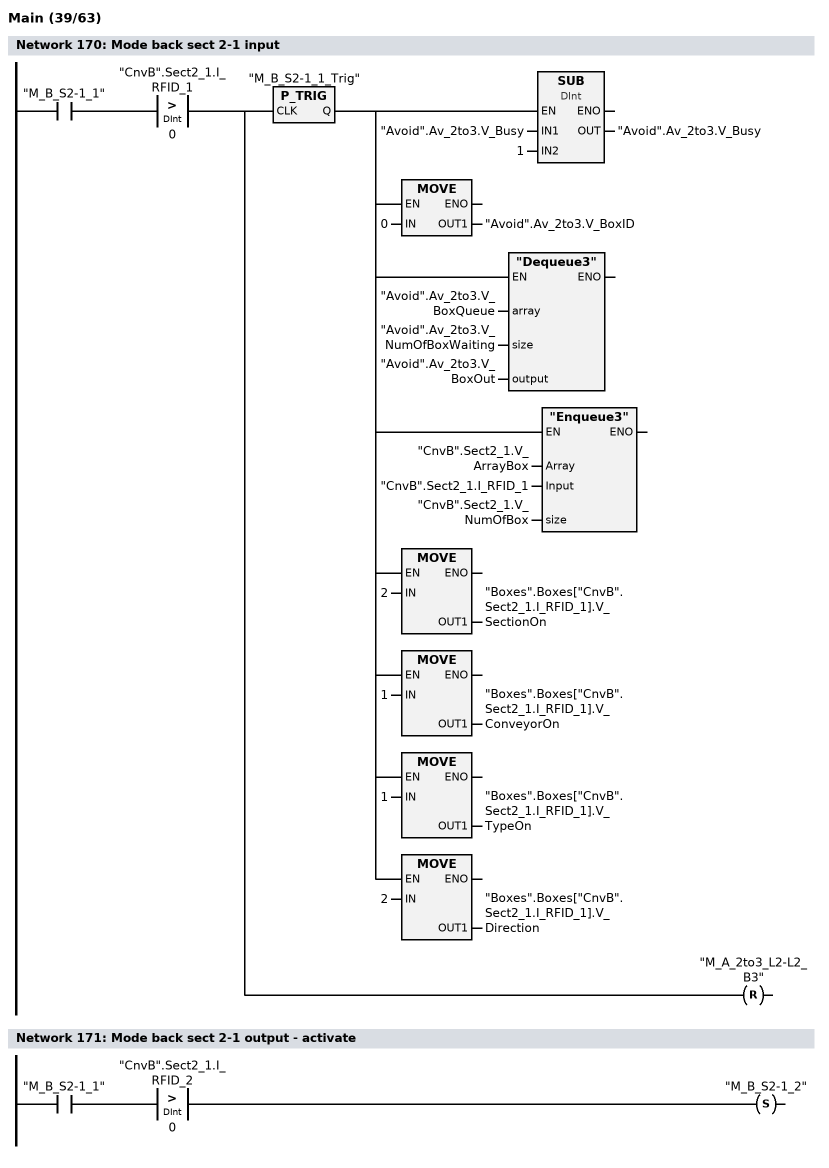
   RUNG wire#powerrail
      Contact( "M_B_S2-1_1" )
      { S7_Templates := "SrcType := DInt" } GT_Contact(in1 := "CnvB".Sect2_1.I_RFID_1, in2 := 0)
      wire#w1
      P_Trig( "M_B_S2-1_1_Trig" )
      wire#w2
      { S7_Templates := "SrcType := DInt" } Sub(in1 := "Avoid".Av_2to3.V_Busy, in2 := 1, out => "Avoid".Av_2to3.V_Busy)
   END_RUNG
   RUNG wire#w2
      Move(in := 0, out1 => "Avoid".Av_2to3.V_BoxID)
   END_RUNG
   RUNG wire#w2
      "Dequeue3"("array" := "Avoid".Av_2to3.V_BoxQueue, size := "Avoid".Av_2to3.V_NumOfBoxWaiting, output := "Avoid".Av_2to3.V_BoxOut)
   END_RUNG
   RUNG wire#w2
      "Enqueue3"("Array" := "CnvB".Sect2_1.V_ArrayBox, Input := "CnvB".Sect2_1.I_RFID_1, size := "CnvB".Sect2_1.V_NumOfBox)
   END_RUNG
   RUNG wire#w2
      Move(in := 2, out1 => "Boxes".Boxes["CnvB".Sect2_1.I_RFID_1].V_SectionOn)
   END_RUNG
   RUNG wire#w2
      Move(in := 1, out1 => "Boxes".Boxes["CnvB".Sect2_1.I_RFID_1].V_ConveyorOn)
   END_RUNG
   RUNG wire#w2
      Move(in := 1, out1 => "Boxes".Boxes["CnvB".Sect2_1.I_RFID_1].V_TypeOn)
   END_RUNG
   RUNG wire#w2
      Move(in := 2, out1 => "Boxes".Boxes["CnvB".Sect2_1.I_RFID_1].V_Direction)
   END_RUNG
   RUNG wire#w1
      R_Coil( "M_A_2to3_L2-L2_B3" )
   END_RUNG
   // the same network as SCL:
   #_w1 := "M_B_S2-1_1" AND ("CnvB".Sect2_1.I_RFID_1 > 0);
   #_w2 := #_w1 AND NOT "M_B_S2-1_1_Trig";   // rising edge
   "M_B_S2-1_1_Trig" := #_w1;
   IF #_w2 THEN
       "Avoid".Av_2to3.V_Busy := "Avoid".Av_2to3.V_Busy - 1;
       "Avoid".Av_2to3.V_BoxID := 0;
       "Dequeue3"("array" := "Avoid".Av_2to3.V_BoxQueue,
                  size := "Avoid".Av_2to3.V_NumOfBoxWaiting,
                  output := "Avoid".Av_2to3.V_BoxOut);
       "Enqueue3"("Array" := "CnvB".Sect2_1.V_ArrayBox,
                  Input := "CnvB".Sect2_1.I_RFID_1,
                  size := "CnvB".Sect2_1.V_NumOfBox);
       "Boxes".Boxes["CnvB".Sect2_1.I_RFID_1].V_SectionOn := 2;
       "Boxes".Boxes["CnvB".Sect2_1.I_RFID_1].V_ConveyorOn := 1;
       "Boxes".Boxes["CnvB".Sect2_1.I_RFID_1].V_TypeOn := 1;
       "Boxes".Boxes["CnvB".Sect2_1.I_RFID_1].V_Direction := 2;
   END_IF;
   IF #_w1 THEN "M_A_2to3_L2-L2_B3" := FALSE; END_IF;
END_REGION

REGION Network 171: Mode back sect 2-1 output - activate
   RUNG wire#powerrail
      Contact( "M_B_S2-1_1" )
      { S7_Templates := "SrcType := DInt" } GT_Contact(in1 := "CnvB".Sect2_1.I_RFID_2, in2 := 0)
      S_Coil( "M_B_S2-1_2" )
   END_RUNG
   // the same network as SCL:
   IF "M_B_S2-1_1" AND ("CnvB".Sect2_1.I_RFID_2 > 0) THEN "M_B_S2-1_2" := TRUE; END_IF;
END_REGION

REGION Network 172: Mode back sect 2-1 output
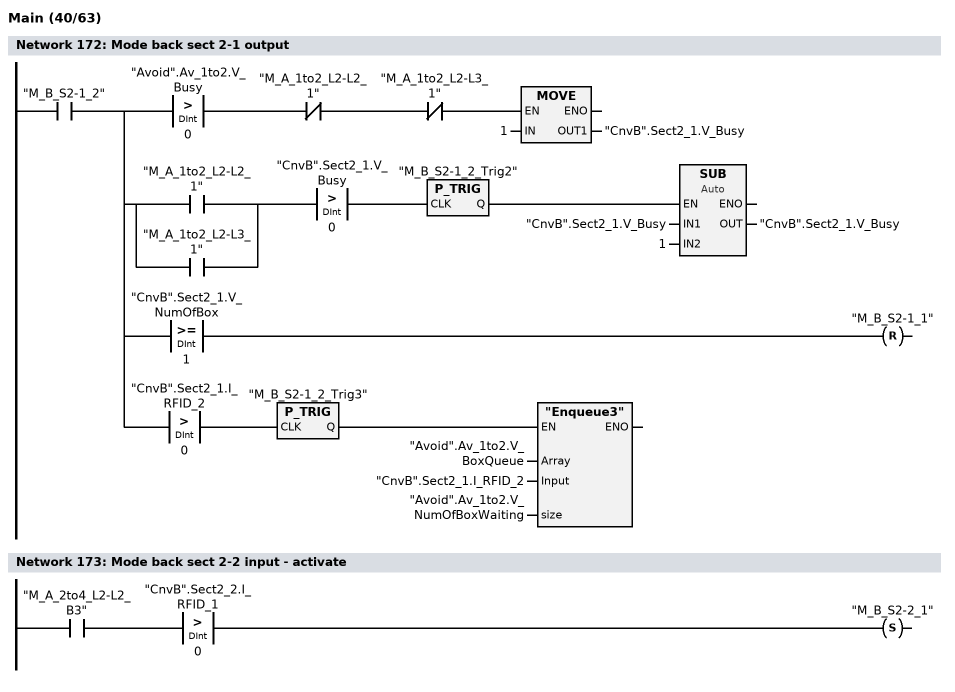
   RUNG wire#powerrail
      Contact( "M_B_S2-1_2" )
      wire#w1
      { S7_Templates := "SrcType := DInt" } GT_Contact(in1 := "Avoid".Av_1to2.V_Busy, in2 := 0)
      I_Contact( "M_A_1to2_L2-L2_1" )
      I_Contact( "M_A_1to2_L2-L3_1" )
      Move(in := 1, out1 => "CnvB".Sect2_1.V_Busy)
   END_RUNG
   RUNG wire#w1
      Contact( "M_A_1to2_L2-L2_1" )
      wire#w2
      { S7_Templates := "SrcType := DInt" } GT_Contact(in1 := "CnvB".Sect2_1.V_Busy, in2 := 0)
      P_Trig( "M_B_S2-1_2_Trig2" )
      Sub(in1 := "CnvB".Sect2_1.V_Busy, in2 := 1, out => "CnvB".Sect2_1.V_Busy)
   END_RUNG
   RUNG wire#w1
      Contact( "M_A_1to2_L2-L3_1" )
   END_RUNG wire#w2
   RUNG wire#w1
      { S7_Templates := "SrcType := DInt" } GE_Contact(in1 := "CnvB".Sect2_1.V_NumOfBox, in2 := 1)
      R_Coil( "M_B_S2-1_1" )
   END_RUNG
   RUNG wire#w1
      { S7_Templates := "SrcType := DInt" } GT_Contact(in1 := "CnvB".Sect2_1.I_RFID_2, in2 := 0)
      P_Trig( "M_B_S2-1_2_Trig3" )
      "Enqueue3"("Array" := "Avoid".Av_1to2.V_BoxQueue, Input := "CnvB".Sect2_1.I_RFID_2, size := "Avoid".Av_1to2.V_NumOfBoxWaiting)
   END_RUNG
   // the same network as SCL:
   IF "M_B_S2-1_2" AND ("Avoid".Av_1to2.V_Busy > 0) AND NOT "M_A_1to2_L2-L2_1" AND NOT "M_A_1to2_L2-L3_1" THEN
       "CnvB".Sect2_1.V_Busy := 1;
   END_IF;
   #_w1 := "M_B_S2-1_2" AND ("M_A_1to2_L2-L2_1" OR "M_A_1to2_L2-L3_1") AND ("CnvB".Sect2_1.V_Busy > 0);
   #_w2 := #_w1 AND NOT "M_B_S2-1_2_Trig2";   // rising edge
   "M_B_S2-1_2_Trig2" := #_w1;
   IF #_w2 THEN "CnvB".Sect2_1.V_Busy := "CnvB".Sect2_1.V_Busy - 1; END_IF;
   IF "M_B_S2-1_2" AND ("CnvB".Sect2_1.V_NumOfBox >= 1) THEN "M_B_S2-1_1" := FALSE; END_IF;
   #_w3 := "M_B_S2-1_2" AND ("CnvB".Sect2_1.I_RFID_2 > 0);
   #_w4 := #_w3 AND NOT "M_B_S2-1_2_Trig3";   // rising edge
   "M_B_S2-1_2_Trig3" := #_w3;
   IF #_w4 THEN
       "Enqueue3"("Array" := "Avoid".Av_1to2.V_BoxQueue,
                  Input := "CnvB".Sect2_1.I_RFID_2,
                  size := "Avoid".Av_1to2.V_NumOfBoxWaiting);
   END_IF;
END_REGION

REGION Network 173: Mode back sect 2-2 input - activate
   RUNG wire#powerrail
      Contact( "M_A_2to4_L2-L2_B3" )
      { S7_Templates := "SrcType := DInt" } GT_Contact(in1 := "CnvB".Sect2_2.I_RFID_1, in2 := 0)
      S_Coil( "M_B_S2-2_1" )
   END_RUNG
   // the same network as SCL:
   IF "M_A_2to4_L2-L2_B3" AND ("CnvB".Sect2_2.I_RFID_1 > 0) THEN "M_B_S2-2_1" := TRUE; END_IF;
END_REGION

REGION Network 174: Mode back sect 2-2 input
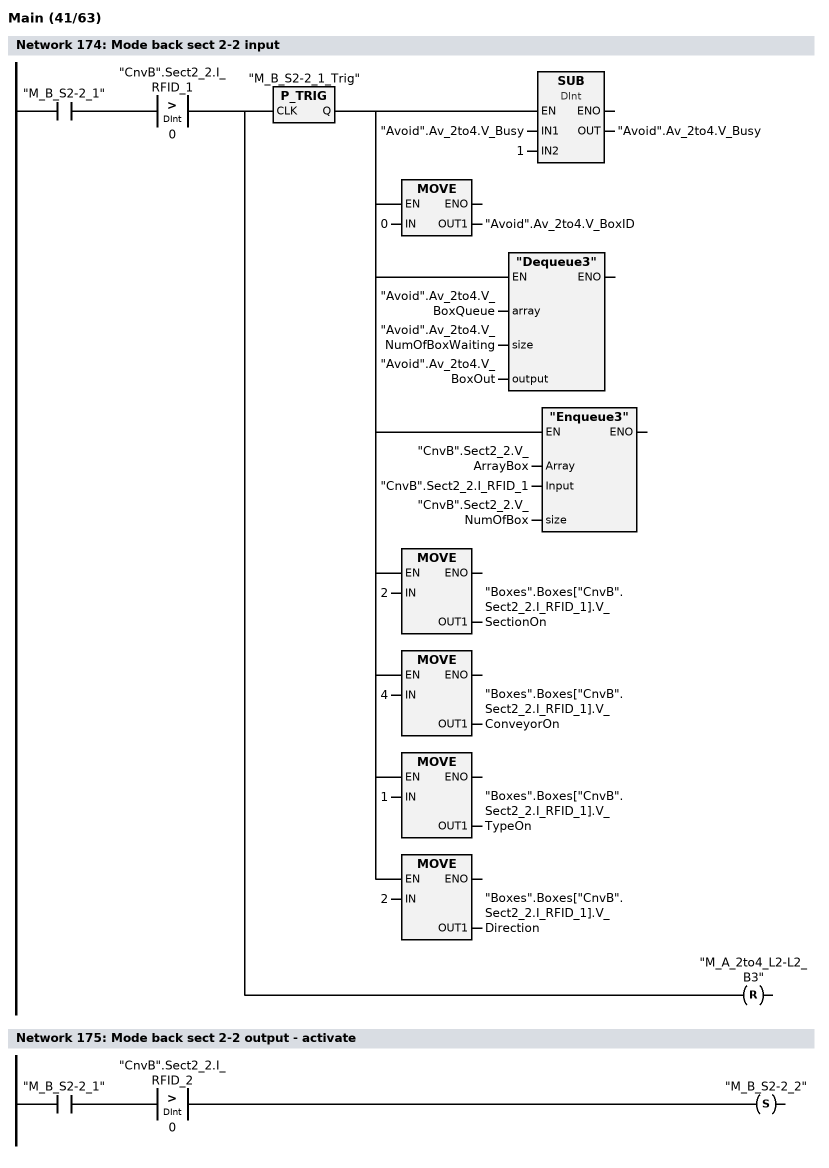
   RUNG wire#powerrail
      Contact( "M_B_S2-2_1" )
      { S7_Templates := "SrcType := DInt" } GT_Contact(in1 := "CnvB".Sect2_2.I_RFID_1, in2 := 0)
      wire#w1
      P_Trig( "M_B_S2-2_1_Trig" )
      wire#w2
      { S7_Templates := "SrcType := DInt" } Sub(in1 := "Avoid".Av_2to4.V_Busy, in2 := 1, out => "Avoid".Av_2to4.V_Busy)
   END_RUNG
   RUNG wire#w2
      Move(in := 0, out1 => "Avoid".Av_2to4.V_BoxID)
   END_RUNG
   RUNG wire#w2
      "Dequeue3"("array" := "Avoid".Av_2to4.V_BoxQueue, size := "Avoid".Av_2to4.V_NumOfBoxWaiting, output := "Avoid".Av_2to4.V_BoxOut)
   END_RUNG
   RUNG wire#w2
      "Enqueue3"("Array" := "CnvB".Sect2_2.V_ArrayBox, Input := "CnvB".Sect2_2.I_RFID_1, size := "CnvB".Sect2_2.V_NumOfBox)
   END_RUNG
   RUNG wire#w2
      Move(in := 2, out1 => "Boxes".Boxes["CnvB".Sect2_2.I_RFID_1].V_SectionOn)
   END_RUNG
   RUNG wire#w2
      Move(in := 4, out1 => "Boxes".Boxes["CnvB".Sect2_2.I_RFID_1].V_ConveyorOn)
   END_RUNG
   RUNG wire#w2
      Move(in := 1, out1 => "Boxes".Boxes["CnvB".Sect2_2.I_RFID_1].V_TypeOn)
   END_RUNG
   RUNG wire#w2
      Move(in := 2, out1 => "Boxes".Boxes["CnvB".Sect2_2.I_RFID_1].V_Direction)
   END_RUNG
   RUNG wire#w1
      R_Coil( "M_A_2to4_L2-L2_B3" )
   END_RUNG
   // the same network as SCL:
   #_w1 := "M_B_S2-2_1" AND ("CnvB".Sect2_2.I_RFID_1 > 0);
   #_w2 := #_w1 AND NOT "M_B_S2-2_1_Trig";   // rising edge
   "M_B_S2-2_1_Trig" := #_w1;
   IF #_w2 THEN
       "Avoid".Av_2to4.V_Busy := "Avoid".Av_2to4.V_Busy - 1;
       "Avoid".Av_2to4.V_BoxID := 0;
       "Dequeue3"("array" := "Avoid".Av_2to4.V_BoxQueue,
                  size := "Avoid".Av_2to4.V_NumOfBoxWaiting,
                  output := "Avoid".Av_2to4.V_BoxOut);
       "Enqueue3"("Array" := "CnvB".Sect2_2.V_ArrayBox,
                  Input := "CnvB".Sect2_2.I_RFID_1,
                  size := "CnvB".Sect2_2.V_NumOfBox);
       "Boxes".Boxes["CnvB".Sect2_2.I_RFID_1].V_SectionOn := 2;
       "Boxes".Boxes["CnvB".Sect2_2.I_RFID_1].V_ConveyorOn := 4;
       "Boxes".Boxes["CnvB".Sect2_2.I_RFID_1].V_TypeOn := 1;
       "Boxes".Boxes["CnvB".Sect2_2.I_RFID_1].V_Direction := 2;
   END_IF;
   IF #_w1 THEN "M_A_2to4_L2-L2_B3" := FALSE; END_IF;
END_REGION

REGION Network 175: Mode back sect 2-2 output - activate
   RUNG wire#powerrail
      Contact( "M_B_S2-2_1" )
      { S7_Templates := "SrcType := DInt" } GT_Contact(in1 := "CnvB".Sect2_2.I_RFID_2, in2 := 0)
      S_Coil( "M_B_S2-2_2" )
   END_RUNG
   // the same network as SCL:
   IF "M_B_S2-2_1" AND ("CnvB".Sect2_2.I_RFID_2 > 0) THEN "M_B_S2-2_2" := TRUE; END_IF;
END_REGION

REGION Network 176: Mode back sect 2-2 output
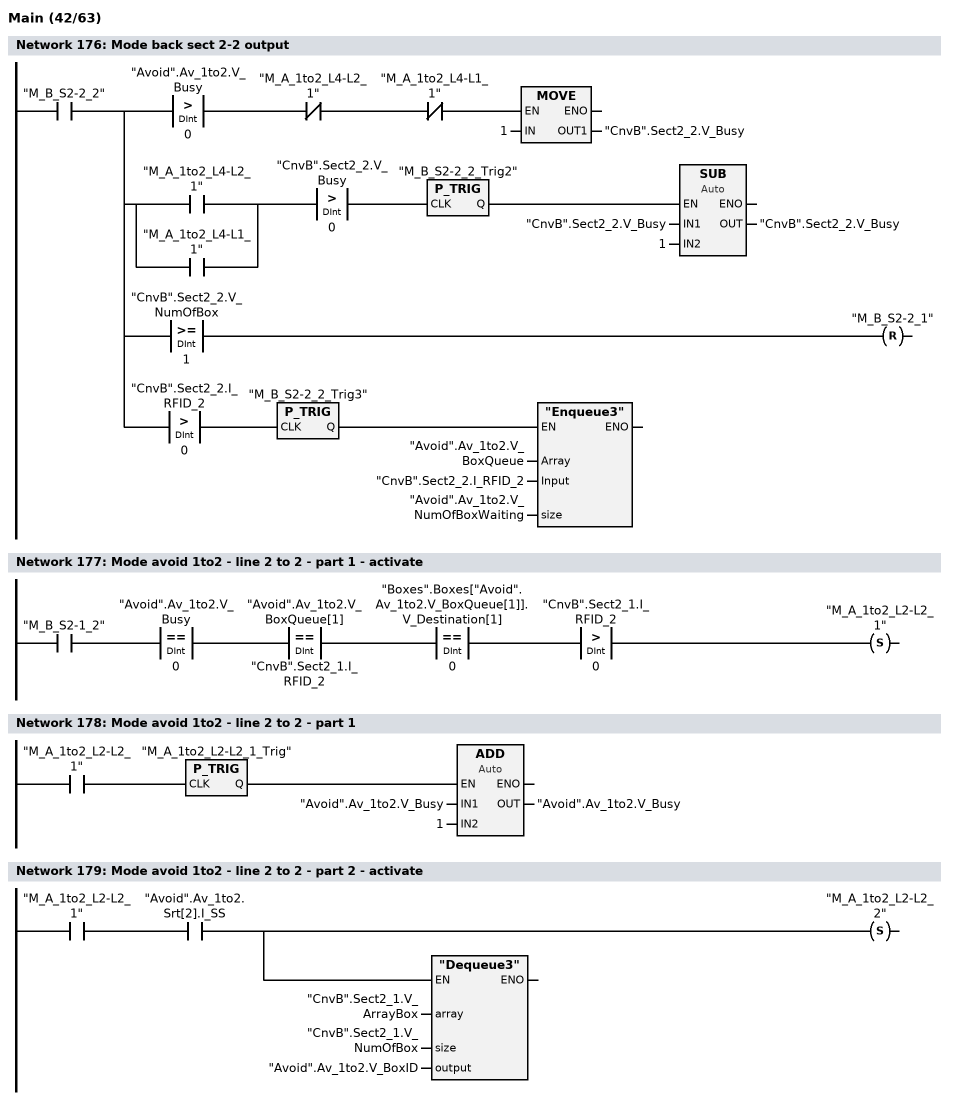
   RUNG wire#powerrail
      Contact( "M_B_S2-2_2" )
      wire#w1
      { S7_Templates := "SrcType := DInt" } GT_Contact(in1 := "Avoid".Av_1to2.V_Busy, in2 := 0)
      I_Contact( "M_A_1to2_L4-L2_1" )
      I_Contact( "M_A_1to2_L4-L1_1" )
      Move(in := 1, out1 => "CnvB".Sect2_2.V_Busy)
   END_RUNG
   RUNG wire#w1
      Contact( "M_A_1to2_L4-L2_1" )
      wire#w2
      { S7_Templates := "SrcType := DInt" } GT_Contact(in1 := "CnvB".Sect2_2.V_Busy, in2 := 0)
      P_Trig( "M_B_S2-2_2_Trig2" )
      Sub(in1 := "CnvB".Sect2_2.V_Busy, in2 := 1, out => "CnvB".Sect2_2.V_Busy)
   END_RUNG
   RUNG wire#w1
      Contact( "M_A_1to2_L4-L1_1" )
   END_RUNG wire#w2
   RUNG wire#w1
      { S7_Templates := "SrcType := DInt" } GE_Contact(in1 := "CnvB".Sect2_2.V_NumOfBox, in2 := 1)
      R_Coil( "M_B_S2-2_1" )
   END_RUNG
   RUNG wire#w1
      { S7_Templates := "SrcType := DInt" } GT_Contact(in1 := "CnvB".Sect2_2.I_RFID_2, in2 := 0)
      P_Trig( "M_B_S2-2_2_Trig3" )
      "Enqueue3"("Array" := "Avoid".Av_1to2.V_BoxQueue, Input := "CnvB".Sect2_2.I_RFID_2, size := "Avoid".Av_1to2.V_NumOfBoxWaiting)
   END_RUNG
   // the same network as SCL:
   IF "M_B_S2-2_2" AND ("Avoid".Av_1to2.V_Busy > 0) AND NOT "M_A_1to2_L4-L2_1" AND NOT "M_A_1to2_L4-L1_1" THEN
       "CnvB".Sect2_2.V_Busy := 1;
   END_IF;
   #_w1 := "M_B_S2-2_2" AND ("M_A_1to2_L4-L2_1" OR "M_A_1to2_L4-L1_1") AND ("CnvB".Sect2_2.V_Busy > 0);
   #_w2 := #_w1 AND NOT "M_B_S2-2_2_Trig2";   // rising edge
   "M_B_S2-2_2_Trig2" := #_w1;
   IF #_w2 THEN "CnvB".Sect2_2.V_Busy := "CnvB".Sect2_2.V_Busy - 1; END_IF;
   IF "M_B_S2-2_2" AND ("CnvB".Sect2_2.V_NumOfBox >= 1) THEN "M_B_S2-2_1" := FALSE; END_IF;
   #_w3 := "M_B_S2-2_2" AND ("CnvB".Sect2_2.I_RFID_2 > 0);
   #_w4 := #_w3 AND NOT "M_B_S2-2_2_Trig3";   // rising edge
   "M_B_S2-2_2_Trig3" := #_w3;
   IF #_w4 THEN
       "Enqueue3"("Array" := "Avoid".Av_1to2.V_BoxQueue,
                  Input := "CnvB".Sect2_2.I_RFID_2,
                  size := "Avoid".Av_1to2.V_NumOfBoxWaiting);
   END_IF;
END_REGION

REGION Network 177: Mode avoid 1to2 - line 2 to 2 - part 1 - activate
   RUNG wire#powerrail
      Contact( "M_B_S2-1_2" )
      { S7_Templates := "SrcType := DInt" } EQ_Contact(in1 := "Avoid".Av_1to2.V_Busy, in2 := 0)
      { S7_Templates := "SrcType := DInt" } EQ_Contact(in1 := "Avoid".Av_1to2.V_BoxQueue[1], in2 := "CnvB".Sect2_1.I_RFID_2)
      { S7_Templates := "SrcType := DInt" } EQ_Contact(in1 := "Boxes".Boxes["Avoid".Av_1to2.V_BoxQueue[1]].V_Destination[1], in2 := 0)
      { S7_Templates := "SrcType := DInt" } GT_Contact(in1 := "CnvB".Sect2_1.I_RFID_2, in2 := 0)
      S_Coil( "M_A_1to2_L2-L2_1" )
   END_RUNG
   // the same network as SCL:
   IF "M_B_S2-1_2" AND ("Avoid".Av_1to2.V_Busy = 0) AND ("Avoid".Av_1to2.V_BoxQueue[1] = "CnvB".Sect2_1.I_RFID_2) AND ("Boxes".Boxes["Avoid".Av_1to2.V_BoxQueue[1]].V_Destination[1] = 0) AND ("CnvB".Sect2_1.I_RFID_2 > 0) THEN
       "M_A_1to2_L2-L2_1" := TRUE;
   END_IF;
END_REGION

REGION Network 178: Mode avoid 1to2 - line 2 to 2 - part 1
   RUNG wire#powerrail
      Contact( "M_A_1to2_L2-L2_1" )
      P_Trig( "M_A_1to2_L2-L2_1_Trig" )
      Add(in1 := "Avoid".Av_1to2.V_Busy, in2 := 1, out => "Avoid".Av_1to2.V_Busy)
   END_RUNG
   // the same network as SCL:
   #_w1 := "M_A_1to2_L2-L2_1" AND NOT "M_A_1to2_L2-L2_1_Trig";   // rising edge
   "M_A_1to2_L2-L2_1_Trig" := "M_A_1to2_L2-L2_1";
   IF #_w1 THEN "Avoid".Av_1to2.V_Busy := "Avoid".Av_1to2.V_Busy + 1; END_IF;
END_REGION

REGION Network 179: Mode avoid 1to2 - line 2 to 2 - part 2 - activate
   RUNG wire#powerrail
      Contact( "M_A_1to2_L2-L2_1" )
      Contact( "Avoid".Av_1to2.Srt[2].I_SS )
      wire#w1
      S_Coil( "M_A_1to2_L2-L2_2" )
   END_RUNG
   RUNG wire#w1
      "Dequeue3"("array" := "CnvB".Sect2_1.V_ArrayBox, size := "CnvB".Sect2_1.V_NumOfBox, output := "Avoid".Av_1to2.V_BoxID)
   END_RUNG
   // the same network as SCL:
   IF "M_A_1to2_L2-L2_1" AND "Avoid".Av_1to2.Srt[2].I_SS THEN
       "M_A_1to2_L2-L2_2" := TRUE;
       "Dequeue3"("array" := "CnvB".Sect2_1.V_ArrayBox,
                  size := "CnvB".Sect2_1.V_NumOfBox,
                  output := "Avoid".Av_1to2.V_BoxID);
   END_IF;
END_REGION

REGION Network 180: Mode avoid 1to2 - line 2 to 2 - part 2
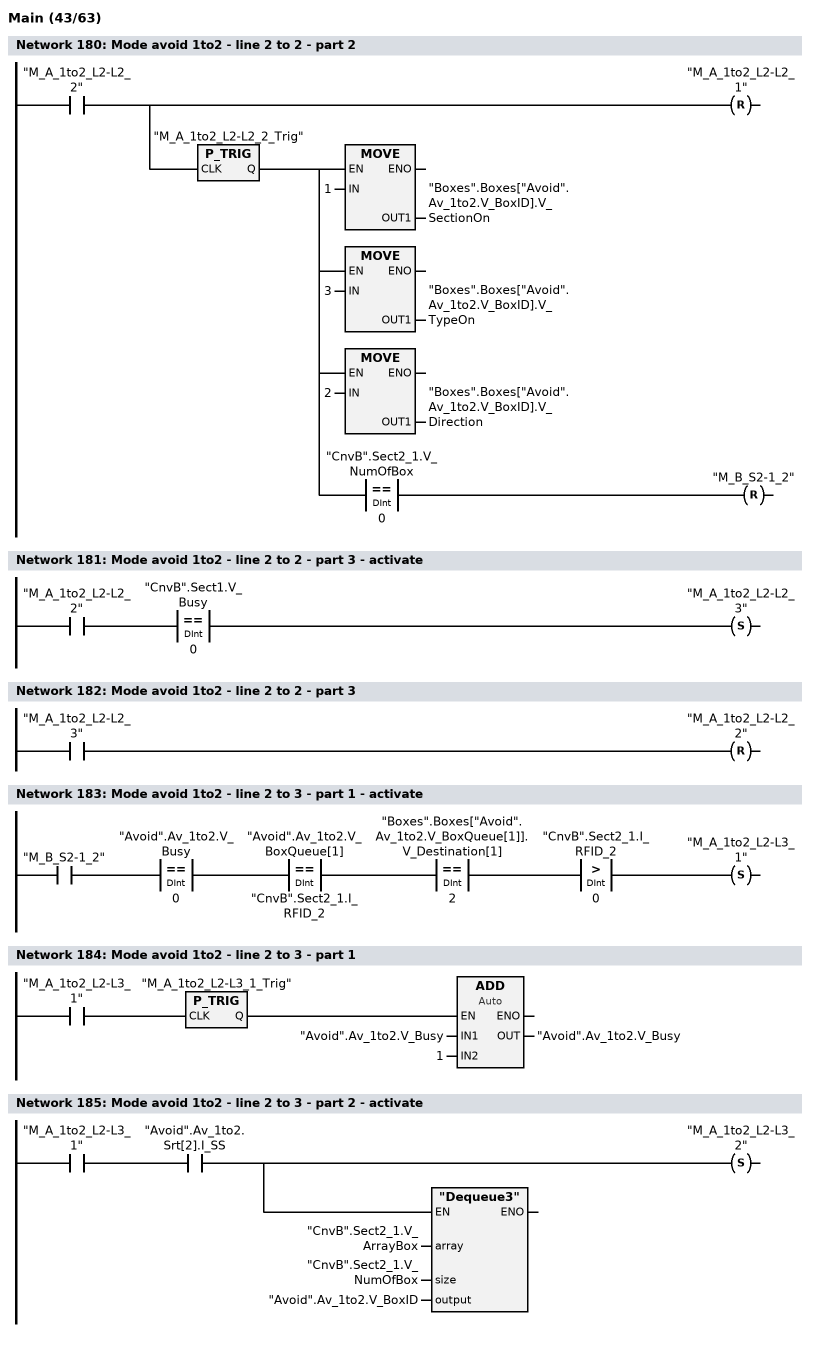
   RUNG wire#powerrail
      Contact( "M_A_1to2_L2-L2_2" )
      wire#w1
      R_Coil( "M_A_1to2_L2-L2_1" )
   END_RUNG
   RUNG wire#w1
      P_Trig( "M_A_1to2_L2-L2_2_Trig" )
      wire#w2
      Move(in := 1, out1 => "Boxes".Boxes["Avoid".Av_1to2.V_BoxID].V_SectionOn)
   END_RUNG
   RUNG wire#w2
      Move(in := 3, out1 => "Boxes".Boxes["Avoid".Av_1to2.V_BoxID].V_TypeOn)
   END_RUNG
   RUNG wire#w2
      Move(in := 2, out1 => "Boxes".Boxes["Avoid".Av_1to2.V_BoxID].V_Direction)
   END_RUNG
   RUNG wire#w2
      { S7_Templates := "SrcType := DInt" } EQ_Contact(in1 := "CnvB".Sect2_1.V_NumOfBox, in2 := 0)
      R_Coil( "M_B_S2-1_2" )
   END_RUNG
   // the same network as SCL:
   IF "M_A_1to2_L2-L2_2" THEN "M_A_1to2_L2-L2_1" := FALSE; END_IF;
   #_w1 := "M_A_1to2_L2-L2_2" AND NOT "M_A_1to2_L2-L2_2_Trig";   // rising edge
   "M_A_1to2_L2-L2_2_Trig" := "M_A_1to2_L2-L2_2";
   IF #_w1 THEN
       "Boxes".Boxes["Avoid".Av_1to2.V_BoxID].V_SectionOn := 1;
       "Boxes".Boxes["Avoid".Av_1to2.V_BoxID].V_TypeOn := 3;
       "Boxes".Boxes["Avoid".Av_1to2.V_BoxID].V_Direction := 2;
   END_IF;
   IF #_w1 AND ("CnvB".Sect2_1.V_NumOfBox = 0) THEN "M_B_S2-1_2" := FALSE; END_IF;
END_REGION

REGION Network 181: Mode avoid 1to2 - line 2 to 2 - part 3 - activate
   RUNG wire#powerrail
      Contact( "M_A_1to2_L2-L2_2" )
      { S7_Templates := "SrcType := DInt" } EQ_Contact(in1 := "CnvB".Sect1.V_Busy, in2 := 0)
      S_Coil( "M_A_1to2_L2-L2_3" )
   END_RUNG
   // the same network as SCL:
   IF "M_A_1to2_L2-L2_2" AND ("CnvB".Sect1.V_Busy = 0) THEN "M_A_1to2_L2-L2_3" := TRUE; END_IF;
END_REGION

REGION Network 182: Mode avoid 1to2 - line 2 to 2 - part 3
   RUNG wire#powerrail
      Contact( "M_A_1to2_L2-L2_3" )
      R_Coil( "M_A_1to2_L2-L2_2" )
   END_RUNG
   // the same network as SCL:
   IF "M_A_1to2_L2-L2_3" THEN "M_A_1to2_L2-L2_2" := FALSE; END_IF;
END_REGION

REGION Network 183: Mode avoid 1to2 - line 2 to 3 - part 1 - activate
   RUNG wire#powerrail
      Contact( "M_B_S2-1_2" )
      { S7_Templates := "SrcType := DInt" } EQ_Contact(in1 := "Avoid".Av_1to2.V_Busy, in2 := 0)
      { S7_Templates := "SrcType := DInt" } EQ_Contact(in1 := "Avoid".Av_1to2.V_BoxQueue[1], in2 := "CnvB".Sect2_1.I_RFID_2)
      { S7_Templates := "SrcType := DInt" } EQ_Contact(in1 := "Boxes".Boxes["Avoid".Av_1to2.V_BoxQueue[1]].V_Destination[1], in2 := 2)
      { S7_Templates := "SrcType := DInt" } GT_Contact(in1 := "CnvB".Sect2_1.I_RFID_2, in2 := 0)
      S_Coil( "M_A_1to2_L2-L3_1" )
   END_RUNG
   // the same network as SCL:
   IF "M_B_S2-1_2" AND ("Avoid".Av_1to2.V_Busy = 0) AND ("Avoid".Av_1to2.V_BoxQueue[1] = "CnvB".Sect2_1.I_RFID_2) AND ("Boxes".Boxes["Avoid".Av_1to2.V_BoxQueue[1]].V_Destination[1] = 2) AND ("CnvB".Sect2_1.I_RFID_2 > 0) THEN
       "M_A_1to2_L2-L3_1" := TRUE;
   END_IF;
END_REGION

REGION Network 184: Mode avoid 1to2 - line 2 to 3 - part 1
   RUNG wire#powerrail
      Contact( "M_A_1to2_L2-L3_1" )
      P_Trig( "M_A_1to2_L2-L3_1_Trig" )
      Add(in1 := "Avoid".Av_1to2.V_Busy, in2 := 1, out => "Avoid".Av_1to2.V_Busy)
   END_RUNG
   // the same network as SCL:
   #_w1 := "M_A_1to2_L2-L3_1" AND NOT "M_A_1to2_L2-L3_1_Trig";   // rising edge
   "M_A_1to2_L2-L3_1_Trig" := "M_A_1to2_L2-L3_1";
   IF #_w1 THEN "Avoid".Av_1to2.V_Busy := "Avoid".Av_1to2.V_Busy + 1; END_IF;
END_REGION

REGION Network 185: Mode avoid 1to2 - line 2 to 3 - part 2 - activate
   RUNG wire#powerrail
      Contact( "M_A_1to2_L2-L3_1" )
      Contact( "Avoid".Av_1to2.Srt[2].I_SS )
      wire#w1
      S_Coil( "M_A_1to2_L2-L3_2" )
   END_RUNG
   RUNG wire#w1
      "Dequeue3"("array" := "CnvB".Sect2_1.V_ArrayBox, size := "CnvB".Sect2_1.V_NumOfBox, output := "Avoid".Av_1to2.V_BoxID)
   END_RUNG
   // the same network as SCL:
   IF "M_A_1to2_L2-L3_1" AND "Avoid".Av_1to2.Srt[2].I_SS THEN
       "M_A_1to2_L2-L3_2" := TRUE;
       "Dequeue3"("array" := "CnvB".Sect2_1.V_ArrayBox,
                  size := "CnvB".Sect2_1.V_NumOfBox,
                  output := "Avoid".Av_1to2.V_BoxID);
   END_IF;
END_REGION

REGION Network 186: Mode avoid 1to2 - line 2 to 3 - part 3
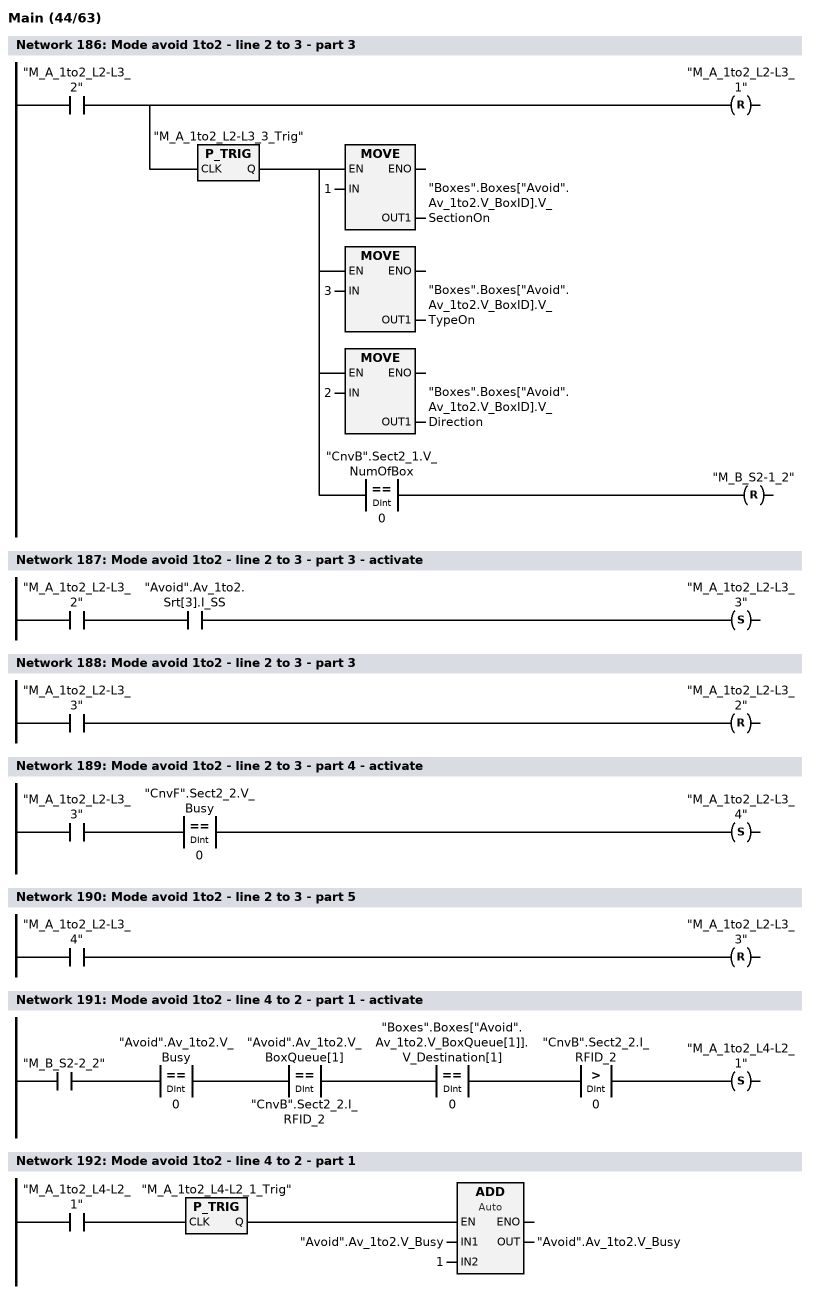
   RUNG wire#powerrail
      Contact( "M_A_1to2_L2-L3_2" )
      wire#w1
      R_Coil( "M_A_1to2_L2-L3_1" )
   END_RUNG
   RUNG wire#w1
      P_Trig( "M_A_1to2_L2-L3_3_Trig" )
      wire#w2
      Move(in := 1, out1 => "Boxes".Boxes["Avoid".Av_1to2.V_BoxID].V_SectionOn)
   END_RUNG
   RUNG wire#w2
      Move(in := 3, out1 => "Boxes".Boxes["Avoid".Av_1to2.V_BoxID].V_TypeOn)
   END_RUNG
   RUNG wire#w2
      Move(in := 2, out1 => "Boxes".Boxes["Avoid".Av_1to2.V_BoxID].V_Direction)
   END_RUNG
   RUNG wire#w2
      { S7_Templates := "SrcType := DInt" } EQ_Contact(in1 := "CnvB".Sect2_1.V_NumOfBox, in2 := 0)
      R_Coil( "M_B_S2-1_2" )
   END_RUNG
   // the same network as SCL:
   IF "M_A_1to2_L2-L3_2" THEN "M_A_1to2_L2-L3_1" := FALSE; END_IF;
   #_w1 := "M_A_1to2_L2-L3_2" AND NOT "M_A_1to2_L2-L3_3_Trig";   // rising edge
   "M_A_1to2_L2-L3_3_Trig" := "M_A_1to2_L2-L3_2";
   IF #_w1 THEN
       "Boxes".Boxes["Avoid".Av_1to2.V_BoxID].V_SectionOn := 1;
       "Boxes".Boxes["Avoid".Av_1to2.V_BoxID].V_TypeOn := 3;
       "Boxes".Boxes["Avoid".Av_1to2.V_BoxID].V_Direction := 2;
   END_IF;
   IF #_w1 AND ("CnvB".Sect2_1.V_NumOfBox = 0) THEN "M_B_S2-1_2" := FALSE; END_IF;
END_REGION

REGION Network 187: Mode avoid 1to2 - line 2 to 3 - part 3 - activate
   RUNG wire#powerrail
      Contact( "M_A_1to2_L2-L3_2" )
      Contact( "Avoid".Av_1to2.Srt[3].I_SS )
      S_Coil( "M_A_1to2_L2-L3_3" )
   END_RUNG
   // the same network as SCL:
   IF "M_A_1to2_L2-L3_2" AND "Avoid".Av_1to2.Srt[3].I_SS THEN "M_A_1to2_L2-L3_3" := TRUE; END_IF;
END_REGION

REGION Network 188: Mode avoid 1to2 - line 2 to 3 - part 3
   RUNG wire#powerrail
      Contact( "M_A_1to2_L2-L3_3" )
      R_Coil( "M_A_1to2_L2-L3_2" )
   END_RUNG
   // the same network as SCL:
   IF "M_A_1to2_L2-L3_3" THEN "M_A_1to2_L2-L3_2" := FALSE; END_IF;
END_REGION

REGION Network 189: Mode avoid 1to2 - line 2 to 3 - part 4 - activate
   RUNG wire#powerrail
      Contact( "M_A_1to2_L2-L3_3" )
      { S7_Templates := "SrcType := DInt" } EQ_Contact(in1 := "CnvF".Sect2_2.V_Busy, in2 := 0)
      S_Coil( "M_A_1to2_L2-L3_4" )
   END_RUNG
   // the same network as SCL:
   IF "M_A_1to2_L2-L3_3" AND ("CnvF".Sect2_2.V_Busy = 0) THEN "M_A_1to2_L2-L3_4" := TRUE; END_IF;
END_REGION

REGION Network 190: Mode avoid 1to2 - line 2 to 3 - part 5
   RUNG wire#powerrail
      Contact( "M_A_1to2_L2-L3_4" )
      R_Coil( "M_A_1to2_L2-L3_3" )
   END_RUNG
   // the same network as SCL:
   IF "M_A_1to2_L2-L3_4" THEN "M_A_1to2_L2-L3_3" := FALSE; END_IF;
END_REGION

REGION Network 191: Mode avoid 1to2 - line 4 to 2 - part 1 - activate
   RUNG wire#powerrail
      Contact( "M_B_S2-2_2" )
      { S7_Templates := "SrcType := DInt" } EQ_Contact(in1 := "Avoid".Av_1to2.V_Busy, in2 := 0)
      { S7_Templates := "SrcType := DInt" } EQ_Contact(in1 := "Avoid".Av_1to2.V_BoxQueue[1], in2 := "CnvB".Sect2_2.I_RFID_2)
      { S7_Templates := "SrcType := DInt" } EQ_Contact(in1 := "Boxes".Boxes["Avoid".Av_1to2.V_BoxQueue[1]].V_Destination[1], in2 := 0)
      { S7_Templates := "SrcType := DInt" } GT_Contact(in1 := "CnvB".Sect2_2.I_RFID_2, in2 := 0)
      S_Coil( "M_A_1to2_L4-L2_1" )
   END_RUNG
   // the same network as SCL:
   IF "M_B_S2-2_2" AND ("Avoid".Av_1to2.V_Busy = 0) AND ("Avoid".Av_1to2.V_BoxQueue[1] = "CnvB".Sect2_2.I_RFID_2) AND ("Boxes".Boxes["Avoid".Av_1to2.V_BoxQueue[1]].V_Destination[1] = 0) AND ("CnvB".Sect2_2.I_RFID_2 > 0) THEN
       "M_A_1to2_L4-L2_1" := TRUE;
   END_IF;
END_REGION

REGION Network 192: Mode avoid 1to2 - line 4 to 2 - part 1
   RUNG wire#powerrail
      Contact( "M_A_1to2_L4-L2_1" )
      P_Trig( "M_A_1to2_L4-L2_1_Trig" )
      Add(in1 := "Avoid".Av_1to2.V_Busy, in2 := 1, out => "Avoid".Av_1to2.V_Busy)
   END_RUNG
   // the same network as SCL:
   #_w1 := "M_A_1to2_L4-L2_1" AND NOT "M_A_1to2_L4-L2_1_Trig";   // rising edge
   "M_A_1to2_L4-L2_1_Trig" := "M_A_1to2_L4-L2_1";
   IF #_w1 THEN "Avoid".Av_1to2.V_Busy := "Avoid".Av_1to2.V_Busy + 1; END_IF;
END_REGION

REGION Network 193: Mode avoid 1to2 - line 4 to 2 - part 2 - activate
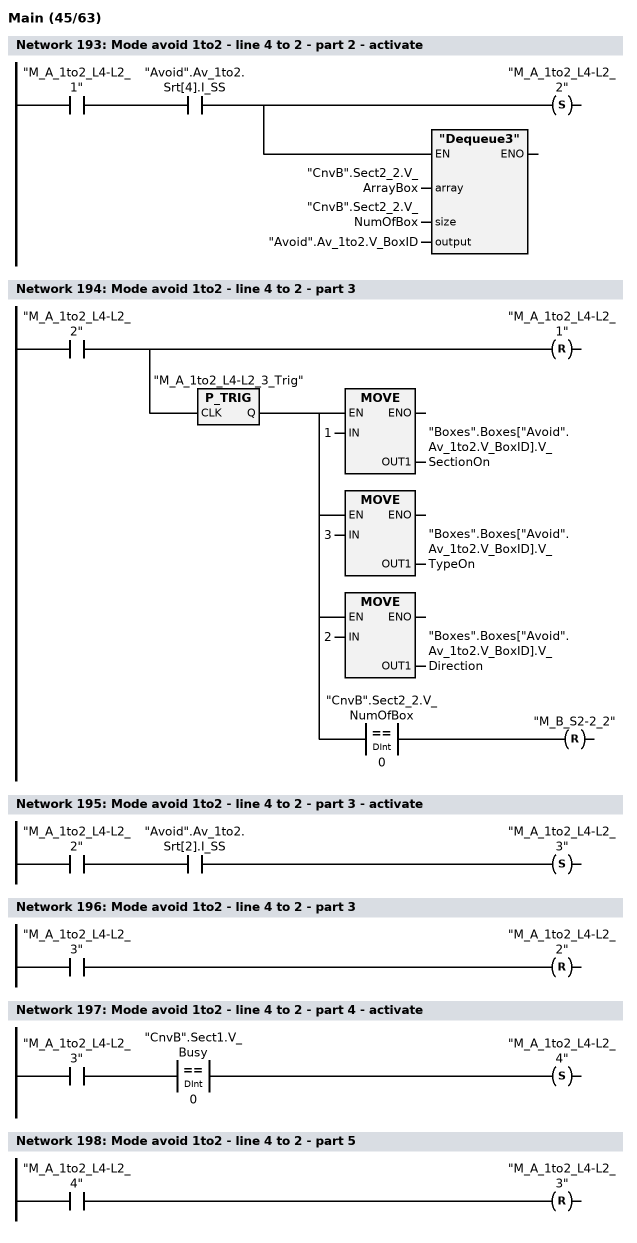
   RUNG wire#powerrail
      Contact( "M_A_1to2_L4-L2_1" )
      Contact( "Avoid".Av_1to2.Srt[4].I_SS )
      wire#w1
      S_Coil( "M_A_1to2_L4-L2_2" )
   END_RUNG
   RUNG wire#w1
      "Dequeue3"("array" := "CnvB".Sect2_2.V_ArrayBox, size := "CnvB".Sect2_2.V_NumOfBox, output := "Avoid".Av_1to2.V_BoxID)
   END_RUNG
   // the same network as SCL:
   IF "M_A_1to2_L4-L2_1" AND "Avoid".Av_1to2.Srt[4].I_SS THEN
       "M_A_1to2_L4-L2_2" := TRUE;
       "Dequeue3"("array" := "CnvB".Sect2_2.V_ArrayBox,
                  size := "CnvB".Sect2_2.V_NumOfBox,
                  output := "Avoid".Av_1to2.V_BoxID);
   END_IF;
END_REGION

REGION Network 194: Mode avoid 1to2 - line 4 to 2 - part 3
   RUNG wire#powerrail
      Contact( "M_A_1to2_L4-L2_2" )
      wire#w1
      R_Coil( "M_A_1to2_L4-L2_1" )
   END_RUNG
   RUNG wire#w1
      P_Trig( "M_A_1to2_L4-L2_3_Trig" )
      wire#w2
      Move(in := 1, out1 => "Boxes".Boxes["Avoid".Av_1to2.V_BoxID].V_SectionOn)
   END_RUNG
   RUNG wire#w2
      Move(in := 3, out1 => "Boxes".Boxes["Avoid".Av_1to2.V_BoxID].V_TypeOn)
   END_RUNG
   RUNG wire#w2
      Move(in := 2, out1 => "Boxes".Boxes["Avoid".Av_1to2.V_BoxID].V_Direction)
   END_RUNG
   RUNG wire#w2
      { S7_Templates := "SrcType := DInt" } EQ_Contact(in1 := "CnvB".Sect2_2.V_NumOfBox, in2 := 0)
      R_Coil( "M_B_S2-2_2" )
   END_RUNG
   // the same network as SCL:
   IF "M_A_1to2_L4-L2_2" THEN "M_A_1to2_L4-L2_1" := FALSE; END_IF;
   #_w1 := "M_A_1to2_L4-L2_2" AND NOT "M_A_1to2_L4-L2_3_Trig";   // rising edge
   "M_A_1to2_L4-L2_3_Trig" := "M_A_1to2_L4-L2_2";
   IF #_w1 THEN
       "Boxes".Boxes["Avoid".Av_1to2.V_BoxID].V_SectionOn := 1;
       "Boxes".Boxes["Avoid".Av_1to2.V_BoxID].V_TypeOn := 3;
       "Boxes".Boxes["Avoid".Av_1to2.V_BoxID].V_Direction := 2;
   END_IF;
   IF #_w1 AND ("CnvB".Sect2_2.V_NumOfBox = 0) THEN "M_B_S2-2_2" := FALSE; END_IF;
END_REGION

REGION Network 195: Mode avoid 1to2 - line 4 to 2 - part 3 - activate
   RUNG wire#powerrail
      Contact( "M_A_1to2_L4-L2_2" )
      Contact( "Avoid".Av_1to2.Srt[2].I_SS )
      S_Coil( "M_A_1to2_L4-L2_3" )
   END_RUNG
   // the same network as SCL:
   IF "M_A_1to2_L4-L2_2" AND "Avoid".Av_1to2.Srt[2].I_SS THEN "M_A_1to2_L4-L2_3" := TRUE; END_IF;
END_REGION

REGION Network 196: Mode avoid 1to2 - line 4 to 2 - part 3
   RUNG wire#powerrail
      Contact( "M_A_1to2_L4-L2_3" )
      R_Coil( "M_A_1to2_L4-L2_2" )
   END_RUNG
   // the same network as SCL:
   IF "M_A_1to2_L4-L2_3" THEN "M_A_1to2_L4-L2_2" := FALSE; END_IF;
END_REGION

REGION Network 197: Mode avoid 1to2 - line 4 to 2 - part 4 - activate
   RUNG wire#powerrail
      Contact( "M_A_1to2_L4-L2_3" )
      { S7_Templates := "SrcType := DInt" } EQ_Contact(in1 := "CnvB".Sect1.V_Busy, in2 := 0)
      S_Coil( "M_A_1to2_L4-L2_4" )
   END_RUNG
   // the same network as SCL:
   IF "M_A_1to2_L4-L2_3" AND ("CnvB".Sect1.V_Busy = 0) THEN "M_A_1to2_L4-L2_4" := TRUE; END_IF;
END_REGION

REGION Network 198: Mode avoid 1to2 - line 4 to 2 - part 5
   RUNG wire#powerrail
      Contact( "M_A_1to2_L4-L2_4" )
      R_Coil( "M_A_1to2_L4-L2_3" )
   END_RUNG
   // the same network as SCL:
   IF "M_A_1to2_L4-L2_4" THEN "M_A_1to2_L4-L2_3" := FALSE; END_IF;
END_REGION

REGION Network 199: Mode avoid 1to2 - line 4 to 1 - part 1 - activate
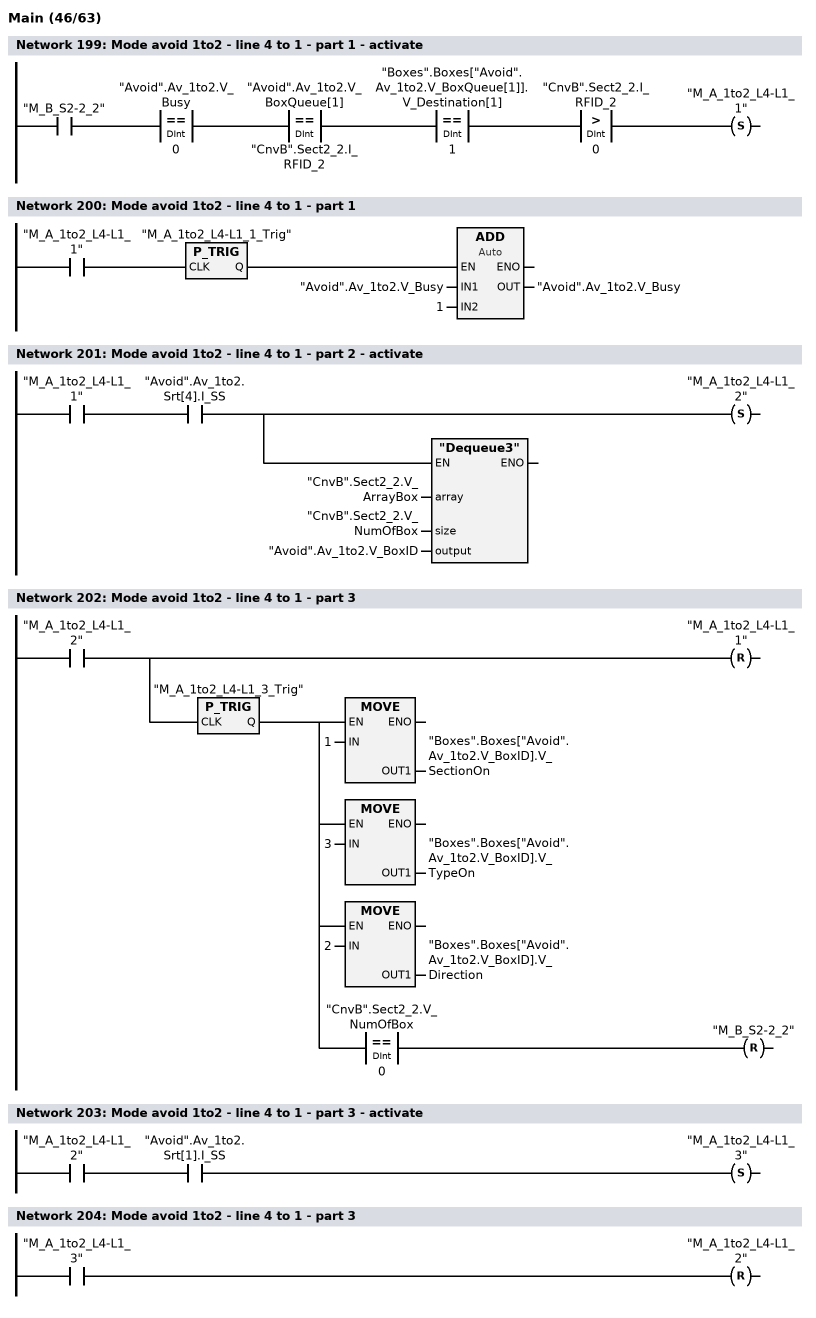
   RUNG wire#powerrail
      Contact( "M_B_S2-2_2" )
      { S7_Templates := "SrcType := DInt" } EQ_Contact(in1 := "Avoid".Av_1to2.V_Busy, in2 := 0)
      { S7_Templates := "SrcType := DInt" } EQ_Contact(in1 := "Avoid".Av_1to2.V_BoxQueue[1], in2 := "CnvB".Sect2_2.I_RFID_2)
      { S7_Templates := "SrcType := DInt" } EQ_Contact(in1 := "Boxes".Boxes["Avoid".Av_1to2.V_BoxQueue[1]].V_Destination[1], in2 := 1)
      { S7_Templates := "SrcType := DInt" } GT_Contact(in1 := "CnvB".Sect2_2.I_RFID_2, in2 := 0)
      S_Coil( "M_A_1to2_L4-L1_1" )
   END_RUNG
   // the same network as SCL:
   IF "M_B_S2-2_2" AND ("Avoid".Av_1to2.V_Busy = 0) AND ("Avoid".Av_1to2.V_BoxQueue[1] = "CnvB".Sect2_2.I_RFID_2) AND ("Boxes".Boxes["Avoid".Av_1to2.V_BoxQueue[1]].V_Destination[1] = 1) AND ("CnvB".Sect2_2.I_RFID_2 > 0) THEN
       "M_A_1to2_L4-L1_1" := TRUE;
   END_IF;
END_REGION

REGION Network 200: Mode avoid 1to2 - line 4 to 1 - part 1
   RUNG wire#powerrail
      Contact( "M_A_1to2_L4-L1_1" )
      P_Trig( "M_A_1to2_L4-L1_1_Trig" )
      Add(in1 := "Avoid".Av_1to2.V_Busy, in2 := 1, out => "Avoid".Av_1to2.V_Busy)
   END_RUNG
   // the same network as SCL:
   #_w1 := "M_A_1to2_L4-L1_1" AND NOT "M_A_1to2_L4-L1_1_Trig";   // rising edge
   "M_A_1to2_L4-L1_1_Trig" := "M_A_1to2_L4-L1_1";
   IF #_w1 THEN "Avoid".Av_1to2.V_Busy := "Avoid".Av_1to2.V_Busy + 1; END_IF;
END_REGION

REGION Network 201: Mode avoid 1to2 - line 4 to 1 - part 2 - activate
   RUNG wire#powerrail
      Contact( "M_A_1to2_L4-L1_1" )
      Contact( "Avoid".Av_1to2.Srt[4].I_SS )
      wire#w1
      S_Coil( "M_A_1to2_L4-L1_2" )
   END_RUNG
   RUNG wire#w1
      "Dequeue3"("array" := "CnvB".Sect2_2.V_ArrayBox, size := "CnvB".Sect2_2.V_NumOfBox, output := "Avoid".Av_1to2.V_BoxID)
   END_RUNG
   // the same network as SCL:
   IF "M_A_1to2_L4-L1_1" AND "Avoid".Av_1to2.Srt[4].I_SS THEN
       "M_A_1to2_L4-L1_2" := TRUE;
       "Dequeue3"("array" := "CnvB".Sect2_2.V_ArrayBox,
                  size := "CnvB".Sect2_2.V_NumOfBox,
                  output := "Avoid".Av_1to2.V_BoxID);
   END_IF;
END_REGION

REGION Network 202: Mode avoid 1to2 - line 4 to 1 - part 3
   RUNG wire#powerrail
      Contact( "M_A_1to2_L4-L1_2" )
      wire#w1
      R_Coil( "M_A_1to2_L4-L1_1" )
   END_RUNG
   RUNG wire#w1
      P_Trig( "M_A_1to2_L4-L1_3_Trig" )
      wire#w2
      Move(in := 1, out1 => "Boxes".Boxes["Avoid".Av_1to2.V_BoxID].V_SectionOn)
   END_RUNG
   RUNG wire#w2
      Move(in := 3, out1 => "Boxes".Boxes["Avoid".Av_1to2.V_BoxID].V_TypeOn)
   END_RUNG
   RUNG wire#w2
      Move(in := 2, out1 => "Boxes".Boxes["Avoid".Av_1to2.V_BoxID].V_Direction)
   END_RUNG
   RUNG wire#w2
      { S7_Templates := "SrcType := DInt" } EQ_Contact(in1 := "CnvB".Sect2_2.V_NumOfBox, in2 := 0)
      R_Coil( "M_B_S2-2_2" )
   END_RUNG
   // the same network as SCL:
   IF "M_A_1to2_L4-L1_2" THEN "M_A_1to2_L4-L1_1" := FALSE; END_IF;
   #_w1 := "M_A_1to2_L4-L1_2" AND NOT "M_A_1to2_L4-L1_3_Trig";   // rising edge
   "M_A_1to2_L4-L1_3_Trig" := "M_A_1to2_L4-L1_2";
   IF #_w1 THEN
       "Boxes".Boxes["Avoid".Av_1to2.V_BoxID].V_SectionOn := 1;
       "Boxes".Boxes["Avoid".Av_1to2.V_BoxID].V_TypeOn := 3;
       "Boxes".Boxes["Avoid".Av_1to2.V_BoxID].V_Direction := 2;
   END_IF;
   IF #_w1 AND ("CnvB".Sect2_2.V_NumOfBox = 0) THEN "M_B_S2-2_2" := FALSE; END_IF;
END_REGION

REGION Network 203: Mode avoid 1to2 - line 4 to 1 - part 3 - activate
   RUNG wire#powerrail
      Contact( "M_A_1to2_L4-L1_2" )
      Contact( "Avoid".Av_1to2.Srt[1].I_SS )
      S_Coil( "M_A_1to2_L4-L1_3" )
   END_RUNG
   // the same network as SCL:
   IF "M_A_1to2_L4-L1_2" AND "Avoid".Av_1to2.Srt[1].I_SS THEN "M_A_1to2_L4-L1_3" := TRUE; END_IF;
END_REGION

REGION Network 204: Mode avoid 1to2 - line 4 to 1 - part 3
   RUNG wire#powerrail
      Contact( "M_A_1to2_L4-L1_3" )
      R_Coil( "M_A_1to2_L4-L1_2" )
   END_RUNG
   // the same network as SCL:
   IF "M_A_1to2_L4-L1_3" THEN "M_A_1to2_L4-L1_2" := FALSE; END_IF;
END_REGION

REGION Network 205: Mode avoid 1to2 - line 4 to 1 - part 4 - activate
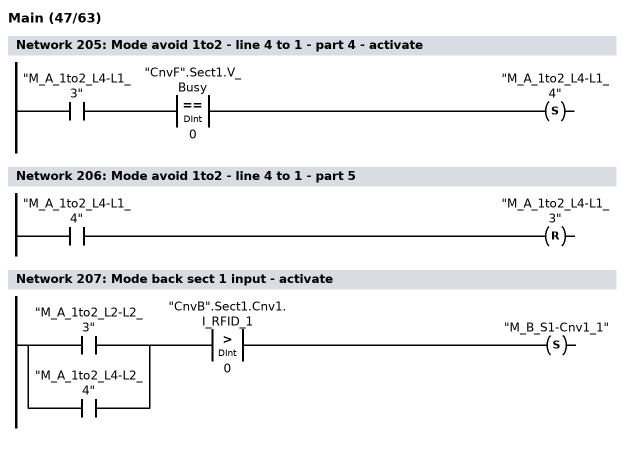
   RUNG wire#powerrail
      Contact( "M_A_1to2_L4-L1_3" )
      { S7_Templates := "SrcType := DInt" } EQ_Contact(in1 := "CnvF".Sect1.V_Busy, in2 := 0)
      S_Coil( "M_A_1to2_L4-L1_4" )
   END_RUNG
   // the same network as SCL:
   IF "M_A_1to2_L4-L1_3" AND ("CnvF".Sect1.V_Busy = 0) THEN "M_A_1to2_L4-L1_4" := TRUE; END_IF;
END_REGION

REGION Network 206: Mode avoid 1to2 - line 4 to 1 - part 5
   RUNG wire#powerrail
      Contact( "M_A_1to2_L4-L1_4" )
      R_Coil( "M_A_1to2_L4-L1_3" )
   END_RUNG
   // the same network as SCL:
   IF "M_A_1to2_L4-L1_4" THEN "M_A_1to2_L4-L1_3" := FALSE; END_IF;
END_REGION

REGION Network 207: Mode back sect 1 input - activate
   RUNG wire#powerrail
      Contact( "M_A_1to2_L2-L2_3" )
      wire#w1
      { S7_Templates := "SrcType := DInt" } GT_Contact(in1 := "CnvB".Sect1.Cnv1.I_RFID_1, in2 := 0)
      S_Coil( "M_B_S1-Cnv1_1" )
   END_RUNG
   RUNG wire#powerrail
      Contact( "M_A_1to2_L4-L2_4" )
   END_RUNG wire#w1
   // the same network as SCL:
   IF ("M_A_1to2_L2-L2_3" OR "M_A_1to2_L4-L2_4") AND ("CnvB".Sect1.Cnv1.I_RFID_1 > 0) THEN
       "M_B_S1-Cnv1_1" := TRUE;
   END_IF;
END_REGION

REGION Network 208: Mode back sect 1 input
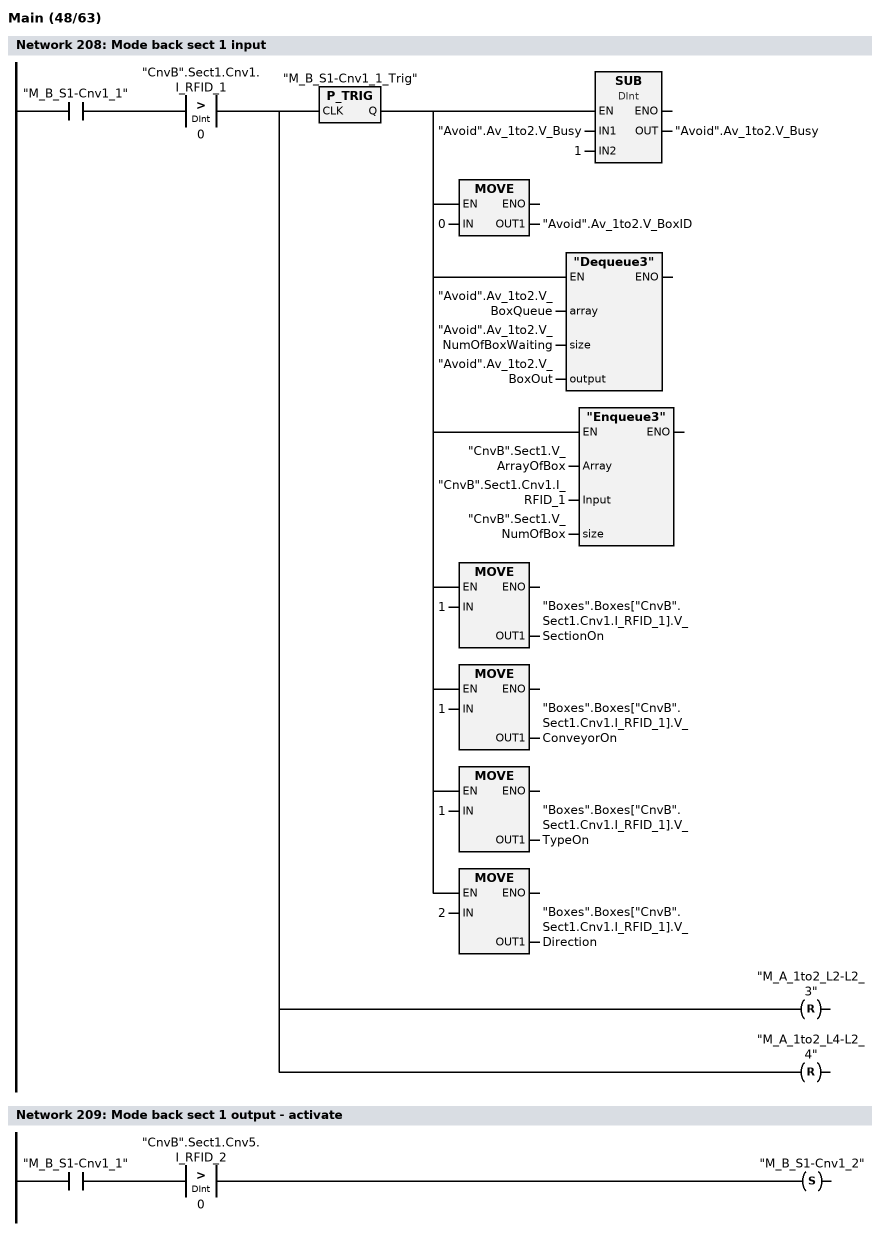
   RUNG wire#powerrail
      Contact( "M_B_S1-Cnv1_1" )
      { S7_Templates := "SrcType := DInt" } GT_Contact(in1 := "CnvB".Sect1.Cnv1.I_RFID_1, in2 := 0)
      wire#w1
      P_Trig( "M_B_S1-Cnv1_1_Trig" )
      wire#w2
      { S7_Templates := "SrcType := DInt" } Sub(in1 := "Avoid".Av_1to2.V_Busy, in2 := 1, out => "Avoid".Av_1to2.V_Busy)
   END_RUNG
   RUNG wire#w2
      Move(in := 0, out1 => "Avoid".Av_1to2.V_BoxID)
   END_RUNG
   RUNG wire#w2
      "Dequeue3"("array" := "Avoid".Av_1to2.V_BoxQueue, size := "Avoid".Av_1to2.V_NumOfBoxWaiting, output := "Avoid".Av_1to2.V_BoxOut)
   END_RUNG
   RUNG wire#w2
      "Enqueue3"("Array" := "CnvB".Sect1.V_ArrayOfBox, Input := "CnvB".Sect1.Cnv1.I_RFID_1, size := "CnvB".Sect1.V_NumOfBox)
   END_RUNG
   RUNG wire#w2
      Move(in := 1, out1 => "Boxes".Boxes["CnvB".Sect1.Cnv1.I_RFID_1].V_SectionOn)
   END_RUNG
   RUNG wire#w2
      Move(in := 1, out1 => "Boxes".Boxes["CnvB".Sect1.Cnv1.I_RFID_1].V_ConveyorOn)
   END_RUNG
   RUNG wire#w2
      Move(in := 1, out1 => "Boxes".Boxes["CnvB".Sect1.Cnv1.I_RFID_1].V_TypeOn)
   END_RUNG
   RUNG wire#w2
      Move(in := 2, out1 => "Boxes".Boxes["CnvB".Sect1.Cnv1.I_RFID_1].V_Direction)
   END_RUNG
   RUNG wire#w1
      R_Coil( "M_A_1to2_L2-L2_3" )
   END_RUNG
   RUNG wire#w1
      R_Coil( "M_A_1to2_L4-L2_4" )
   END_RUNG
   // the same network as SCL:
   #_w1 := "M_B_S1-Cnv1_1" AND ("CnvB".Sect1.Cnv1.I_RFID_1 > 0);
   #_w2 := #_w1 AND NOT "M_B_S1-Cnv1_1_Trig";   // rising edge
   "M_B_S1-Cnv1_1_Trig" := #_w1;
   IF #_w2 THEN
       "Avoid".Av_1to2.V_Busy := "Avoid".Av_1to2.V_Busy - 1;
       "Avoid".Av_1to2.V_BoxID := 0;
       "Dequeue3"("array" := "Avoid".Av_1to2.V_BoxQueue,
                  size := "Avoid".Av_1to2.V_NumOfBoxWaiting,
                  output := "Avoid".Av_1to2.V_BoxOut);
       "Enqueue3"("Array" := "CnvB".Sect1.V_ArrayOfBox,
                  Input := "CnvB".Sect1.Cnv1.I_RFID_1,
                  size := "CnvB".Sect1.V_NumOfBox);
       "Boxes".Boxes["CnvB".Sect1.Cnv1.I_RFID_1].V_SectionOn := 1;
       "Boxes".Boxes["CnvB".Sect1.Cnv1.I_RFID_1].V_ConveyorOn := 1;
       "Boxes".Boxes["CnvB".Sect1.Cnv1.I_RFID_1].V_TypeOn := 1;
       "Boxes".Boxes["CnvB".Sect1.Cnv1.I_RFID_1].V_Direction := 2;
   END_IF;
   IF #_w1 THEN
       "M_A_1to2_L2-L2_3" := FALSE;
       "M_A_1to2_L4-L2_4" := FALSE;
   END_IF;
END_REGION

REGION Network 209: Mode back sect 1 output - activate
   RUNG wire#powerrail
      Contact( "M_B_S1-Cnv1_1" )
      { S7_Templates := "SrcType := DInt" } GT_Contact(in1 := "CnvB".Sect1.Cnv5.I_RFID_2, in2 := 0)
      S_Coil( "M_B_S1-Cnv1_2" )
   END_RUNG
   // the same network as SCL:
   IF "M_B_S1-Cnv1_1" AND ("CnvB".Sect1.Cnv5.I_RFID_2 > 0) THEN "M_B_S1-Cnv1_2" := TRUE; END_IF;
END_REGION

REGION Network 210: Mode back sect 1 output
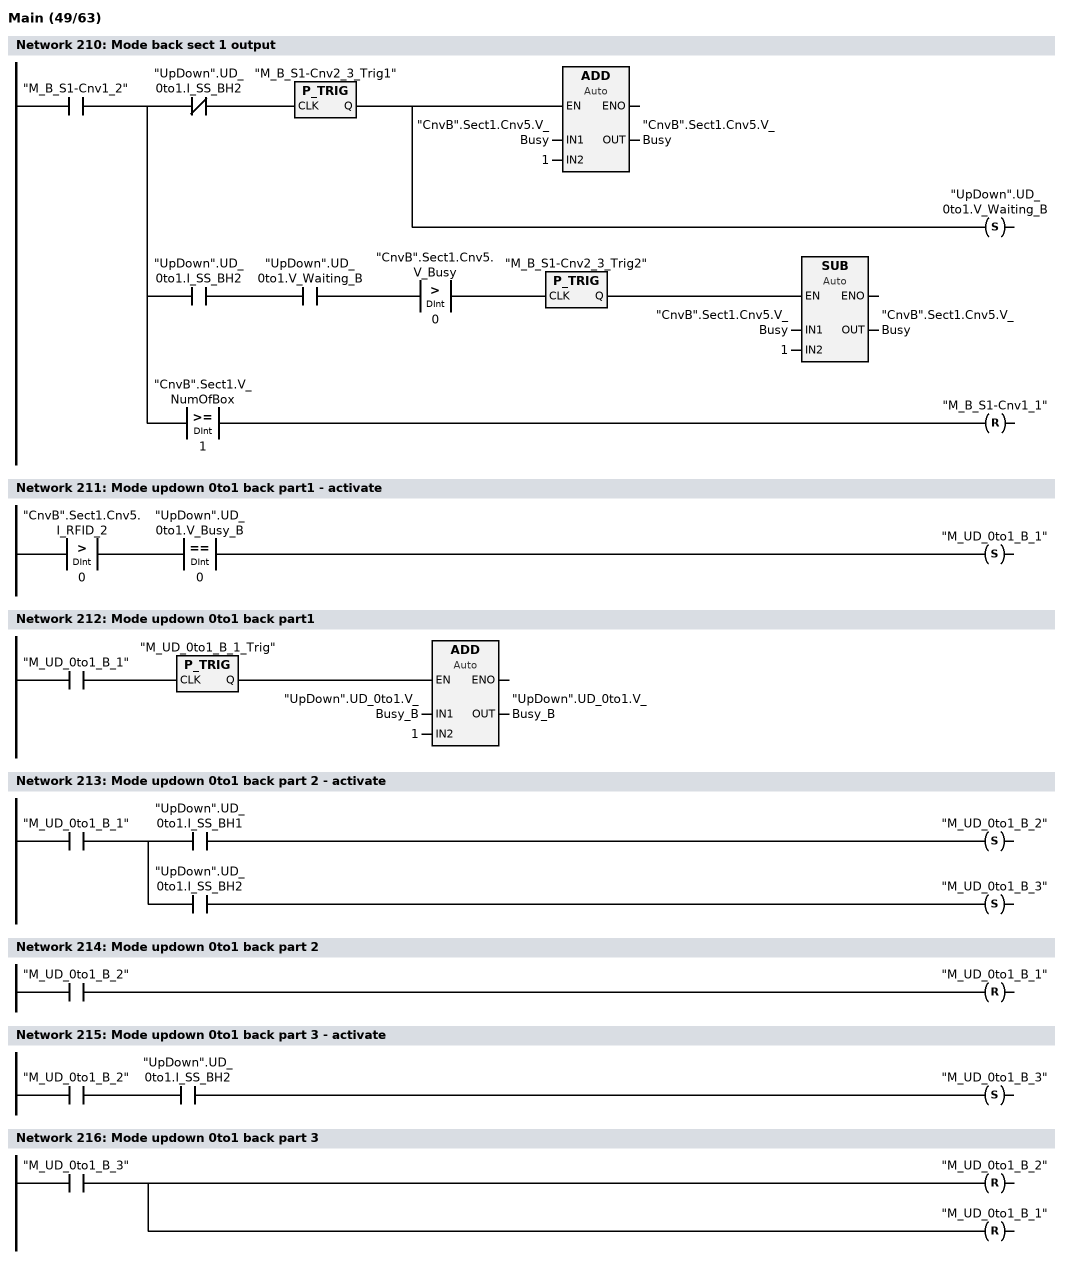
   RUNG wire#powerrail
      Contact( "M_B_S1-Cnv1_2" )
      wire#w1
      I_Contact( "UpDown".UD_0to1.I_SS_BH2 )
      P_Trig( "M_B_S1-Cnv2_3_Trig1" )
      wire#w2
      Add(in1 := "CnvB".Sect1.Cnv5.V_Busy, in2 := 1, out => "CnvB".Sect1.Cnv5.V_Busy)
   END_RUNG
   RUNG wire#w2
      S_Coil( "UpDown".UD_0to1.V_Waiting_B )
   END_RUNG
   RUNG wire#w1
      Contact( "UpDown".UD_0to1.I_SS_BH2 )
      Contact( "UpDown".UD_0to1.V_Waiting_B )
      { S7_Templates := "SrcType := DInt" } GT_Contact(in1 := "CnvB".Sect1.Cnv5.V_Busy, in2 := 0)
      P_Trig( "M_B_S1-Cnv2_3_Trig2" )
      Sub(in1 := "CnvB".Sect1.Cnv5.V_Busy, in2 := 1, out => "CnvB".Sect1.Cnv5.V_Busy)
   END_RUNG
   RUNG wire#w1
      { S7_Templates := "SrcType := DInt" } GE_Contact(in1 := "CnvB".Sect1.V_NumOfBox, in2 := 1)
      R_Coil( "M_B_S1-Cnv1_1" )
   END_RUNG
   // the same network as SCL:
   #_w1 := "M_B_S1-Cnv1_2" AND NOT "UpDown".UD_0to1.I_SS_BH2;
   #_w2 := #_w1 AND NOT "M_B_S1-Cnv2_3_Trig1";   // rising edge
   "M_B_S1-Cnv2_3_Trig1" := #_w1;
   IF #_w2 THEN
       "CnvB".Sect1.Cnv5.V_Busy := "CnvB".Sect1.Cnv5.V_Busy + 1;
       "UpDown".UD_0to1.V_Waiting_B := TRUE;
   END_IF;
   #_w3 := "M_B_S1-Cnv1_2" AND "UpDown".UD_0to1.I_SS_BH2 AND "UpDown".UD_0to1.V_Waiting_B AND ("CnvB".Sect1.Cnv5.V_Busy > 0);
   #_w4 := #_w3 AND NOT "M_B_S1-Cnv2_3_Trig2";   // rising edge
   "M_B_S1-Cnv2_3_Trig2" := #_w3;
   IF #_w4 THEN "CnvB".Sect1.Cnv5.V_Busy := "CnvB".Sect1.Cnv5.V_Busy - 1; END_IF;
   IF "M_B_S1-Cnv1_2" AND ("CnvB".Sect1.V_NumOfBox >= 1) THEN "M_B_S1-Cnv1_1" := FALSE; END_IF;
END_REGION

REGION Network 211: Mode updown 0to1 back part1 - activate
   RUNG wire#powerrail
      { S7_Templates := "SrcType := DInt" } GT_Contact(in1 := "CnvB".Sect1.Cnv5.I_RFID_2, in2 := 0)
      { S7_Templates := "SrcType := DInt" } EQ_Contact(in1 := "UpDown".UD_0to1.V_Busy_B, in2 := 0)
      S_Coil( "M_UD_0to1_B_1" )
   END_RUNG
   // the same network as SCL:
   IF ("CnvB".Sect1.Cnv5.I_RFID_2 > 0) AND ("UpDown".UD_0to1.V_Busy_B = 0) THEN
       "M_UD_0to1_B_1" := TRUE;
   END_IF;
END_REGION

REGION Network 212: Mode updown 0to1 back part1
   RUNG wire#powerrail
      Contact( "M_UD_0to1_B_1" )
      P_Trig( "M_UD_0to1_B_1_Trig" )
      Add(in1 := "UpDown".UD_0to1.V_Busy_B, in2 := 1, out => "UpDown".UD_0to1.V_Busy_B)
   END_RUNG
   // the same network as SCL:
   #_w1 := "M_UD_0to1_B_1" AND NOT "M_UD_0to1_B_1_Trig";   // rising edge
   "M_UD_0to1_B_1_Trig" := "M_UD_0to1_B_1";
   IF #_w1 THEN "UpDown".UD_0to1.V_Busy_B := "UpDown".UD_0to1.V_Busy_B + 1; END_IF;
END_REGION

REGION Network 213: Mode updown 0to1 back part 2 - activate
   RUNG wire#powerrail
      Contact( "M_UD_0to1_B_1" )
      wire#w1
      Contact( "UpDown".UD_0to1.I_SS_BH1 )
      S_Coil( "M_UD_0to1_B_2" )
   END_RUNG
   RUNG wire#w1
      Contact( "UpDown".UD_0to1.I_SS_BH2 )
      S_Coil( "M_UD_0to1_B_3" )
   END_RUNG
   // the same network as SCL:
   IF "M_UD_0to1_B_1" AND "UpDown".UD_0to1.I_SS_BH1 THEN "M_UD_0to1_B_2" := TRUE; END_IF;
   IF "M_UD_0to1_B_1" AND "UpDown".UD_0to1.I_SS_BH2 THEN "M_UD_0to1_B_3" := TRUE; END_IF;
END_REGION

REGION Network 214: Mode updown 0to1 back part 2
   RUNG wire#powerrail
      Contact( "M_UD_0to1_B_2" )
      R_Coil( "M_UD_0to1_B_1" )
   END_RUNG
   // the same network as SCL:
   IF "M_UD_0to1_B_2" THEN "M_UD_0to1_B_1" := FALSE; END_IF;
END_REGION

REGION Network 215: Mode updown 0to1 back part 3 - activate
   RUNG wire#powerrail
      Contact( "M_UD_0to1_B_2" )
      Contact( "UpDown".UD_0to1.I_SS_BH2 )
      S_Coil( "M_UD_0to1_B_3" )
   END_RUNG
   // the same network as SCL:
   IF "M_UD_0to1_B_2" AND "UpDown".UD_0to1.I_SS_BH2 THEN "M_UD_0to1_B_3" := TRUE; END_IF;
END_REGION

REGION Network 216: Mode updown 0to1 back part 3
   RUNG wire#powerrail
      Contact( "M_UD_0to1_B_3" )
      wire#w1
      R_Coil( "M_UD_0to1_B_2" )
   END_RUNG
   RUNG wire#w1
      R_Coil( "M_UD_0to1_B_1" )
   END_RUNG
   // the same network as SCL:
   IF "M_UD_0to1_B_3" THEN
       "M_UD_0to1_B_2" := FALSE;
       "M_UD_0to1_B_1" := FALSE;
   END_IF;
END_REGION

REGION Network 217: Mode updown 0to1 back part 4 - activate
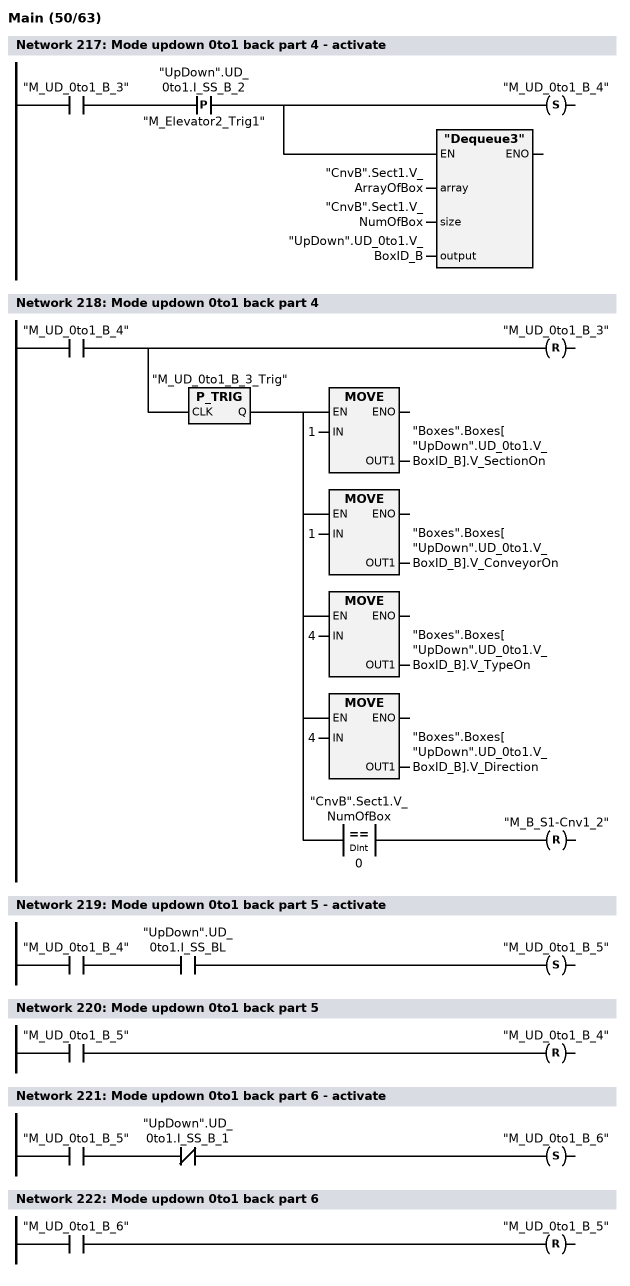
   RUNG wire#powerrail
      Contact( "M_UD_0to1_B_3" )
      P_Contact(operand := "UpDown".UD_0to1.I_SS_B_2, bit := "M_Elevator2_Trig1")
      wire#w1
      S_Coil( "M_UD_0to1_B_4" )
   END_RUNG
   RUNG wire#w1
      "Dequeue3"("array" := "CnvB".Sect1.V_ArrayOfBox, size := "CnvB".Sect1.V_NumOfBox, output := "UpDown".UD_0to1.V_BoxID_B)
   END_RUNG
   // the same network as SCL:
   #_w1 := "M_UD_0to1_B_3" AND "UpDown".UD_0to1.I_SS_B_2 AND NOT "M_Elevator2_Trig1";   // rising edge of "UpDown".UD_0to1.I_SS_B_2
   "M_Elevator2_Trig1" := "UpDown".UD_0to1.I_SS_B_2;
   IF #_w1 THEN
       "M_UD_0to1_B_4" := TRUE;
       "Dequeue3"("array" := "CnvB".Sect1.V_ArrayOfBox,
                  size := "CnvB".Sect1.V_NumOfBox,
                  output := "UpDown".UD_0to1.V_BoxID_B);
   END_IF;
END_REGION

REGION Network 218: Mode updown 0to1 back part 4
   RUNG wire#powerrail
      Contact( "M_UD_0to1_B_4" )
      wire#w1
      R_Coil( "M_UD_0to1_B_3" )
   END_RUNG
   RUNG wire#w1
      P_Trig( "M_UD_0to1_B_3_Trig" )
      wire#w2
      Move(in := 1, out1 => "Boxes".Boxes["UpDown".UD_0to1.V_BoxID_B].V_SectionOn)
   END_RUNG
   RUNG wire#w2
      Move(in := 1, out1 => "Boxes".Boxes["UpDown".UD_0to1.V_BoxID_B].V_ConveyorOn)
   END_RUNG
   RUNG wire#w2
      Move(in := 4, out1 => "Boxes".Boxes["UpDown".UD_0to1.V_BoxID_B].V_TypeOn)
   END_RUNG
   RUNG wire#w2
      Move(in := 4, out1 => "Boxes".Boxes["UpDown".UD_0to1.V_BoxID_B].V_Direction)
   END_RUNG
   RUNG wire#w2
      { S7_Templates := "SrcType := DInt" } EQ_Contact(in1 := "CnvB".Sect1.V_NumOfBox, in2 := 0)
      R_Coil( "M_B_S1-Cnv1_2" )
   END_RUNG
   // the same network as SCL:
   IF "M_UD_0to1_B_4" THEN "M_UD_0to1_B_3" := FALSE; END_IF;
   #_w1 := "M_UD_0to1_B_4" AND NOT "M_UD_0to1_B_3_Trig";   // rising edge
   "M_UD_0to1_B_3_Trig" := "M_UD_0to1_B_4";
   IF #_w1 THEN
       "Boxes".Boxes["UpDown".UD_0to1.V_BoxID_B].V_SectionOn := 1;
       "Boxes".Boxes["UpDown".UD_0to1.V_BoxID_B].V_ConveyorOn := 1;
       "Boxes".Boxes["UpDown".UD_0to1.V_BoxID_B].V_TypeOn := 4;
       "Boxes".Boxes["UpDown".UD_0to1.V_BoxID_B].V_Direction := 4;
   END_IF;
   IF #_w1 AND ("CnvB".Sect1.V_NumOfBox = 0) THEN "M_B_S1-Cnv1_2" := FALSE; END_IF;
END_REGION

REGION Network 219: Mode updown 0to1 back part 5 - activate
   RUNG wire#powerrail
      Contact( "M_UD_0to1_B_4" )
      Contact( "UpDown".UD_0to1.I_SS_BL )
      S_Coil( "M_UD_0to1_B_5" )
   END_RUNG
   // the same network as SCL:
   IF "M_UD_0to1_B_4" AND "UpDown".UD_0to1.I_SS_BL THEN "M_UD_0to1_B_5" := TRUE; END_IF;
END_REGION

REGION Network 220: Mode updown 0to1 back part 5
   RUNG wire#powerrail
      Contact( "M_UD_0to1_B_5" )
      R_Coil( "M_UD_0to1_B_4" )
   END_RUNG
   // the same network as SCL:
   IF "M_UD_0to1_B_5" THEN "M_UD_0to1_B_4" := FALSE; END_IF;
END_REGION

REGION Network 221: Mode updown 0to1 back part 6 - activate
   RUNG wire#powerrail
      Contact( "M_UD_0to1_B_5" )
      I_Contact( "UpDown".UD_0to1.I_SS_B_1 )
      S_Coil( "M_UD_0to1_B_6" )
   END_RUNG
   // the same network as SCL:
   IF "M_UD_0to1_B_5" AND NOT "UpDown".UD_0to1.I_SS_B_1 THEN "M_UD_0to1_B_6" := TRUE; END_IF;
END_REGION

REGION Network 222: Mode updown 0to1 back part 6
   RUNG wire#powerrail
      Contact( "M_UD_0to1_B_6" )
      R_Coil( "M_UD_0to1_B_5" )
   END_RUNG
   // the same network as SCL:
   IF "M_UD_0to1_B_6" THEN "M_UD_0to1_B_5" := FALSE; END_IF;
END_REGION

REGION Network 223: Mode updown 0to1 back part 7 - activate
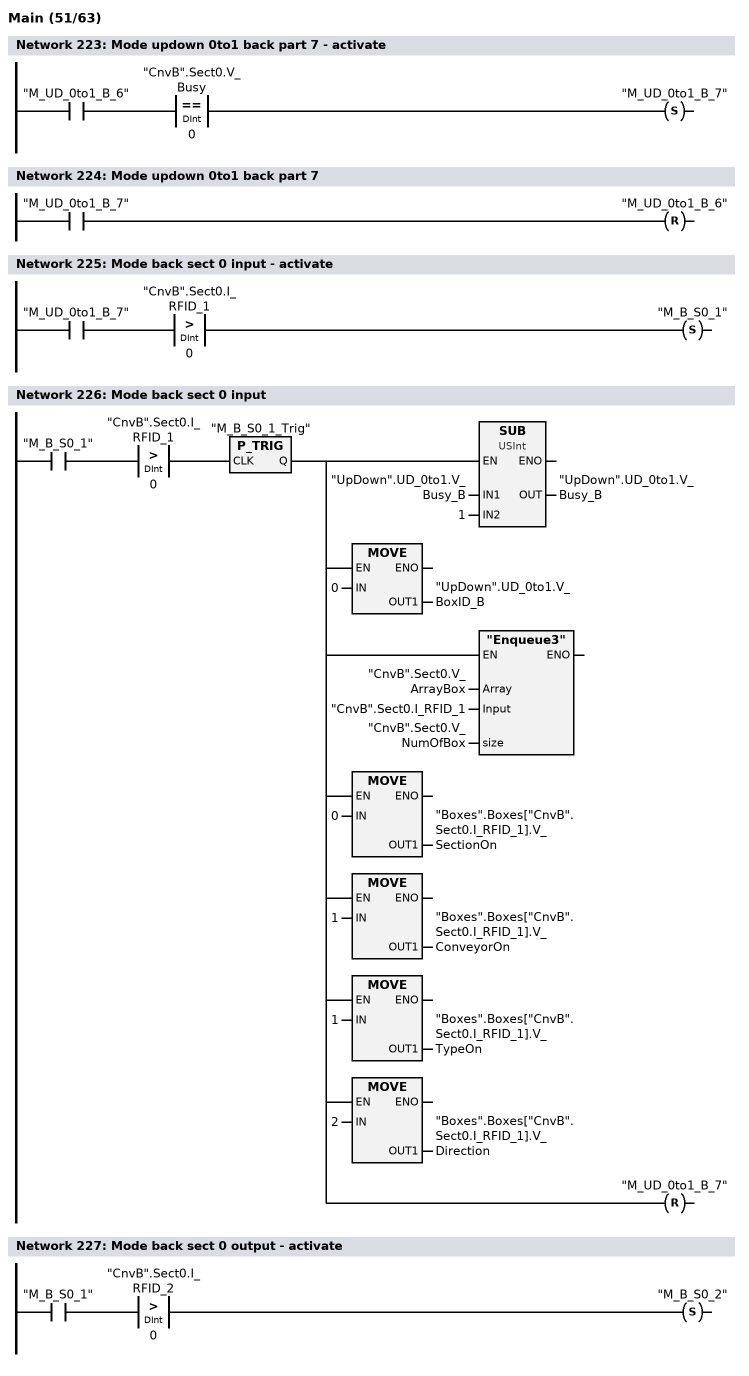
   RUNG wire#powerrail
      Contact( "M_UD_0to1_B_6" )
      { S7_Templates := "SrcType := DInt" } EQ_Contact(in1 := "CnvB".Sect0.V_Busy, in2 := 0)
      S_Coil( "M_UD_0to1_B_7" )
   END_RUNG
   // the same network as SCL:
   IF "M_UD_0to1_B_6" AND ("CnvB".Sect0.V_Busy = 0) THEN "M_UD_0to1_B_7" := TRUE; END_IF;
END_REGION

REGION Network 224: Mode updown 0to1 back part 7
   RUNG wire#powerrail
      Contact( "M_UD_0to1_B_7" )
      R_Coil( "M_UD_0to1_B_6" )
   END_RUNG
   // the same network as SCL:
   IF "M_UD_0to1_B_7" THEN "M_UD_0to1_B_6" := FALSE; END_IF;
END_REGION

REGION Network 225: Mode back sect 0 input - activate
   RUNG wire#powerrail
      Contact( "M_UD_0to1_B_7" )
      { S7_Templates := "SrcType := DInt" } GT_Contact(in1 := "CnvB".Sect0.I_RFID_1, in2 := 0)
      S_Coil( "M_B_S0_1" )
   END_RUNG
   // the same network as SCL:
   IF "M_UD_0to1_B_7" AND ("CnvB".Sect0.I_RFID_1 > 0) THEN "M_B_S0_1" := TRUE; END_IF;
END_REGION

REGION Network 226: Mode back sect 0 input
   RUNG wire#powerrail
      Contact( "M_B_S0_1" )
      { S7_Templates := "SrcType := DInt" } GT_Contact(in1 := "CnvB".Sect0.I_RFID_1, in2 := 0)
      P_Trig( "M_B_S0_1_Trig" )
      wire#w1
      { S7_Templates := "SrcType := USInt" } Sub(in1 := "UpDown".UD_0to1.V_Busy_B, in2 := 1, out => "UpDown".UD_0to1.V_Busy_B)
   END_RUNG
   RUNG wire#w1
      Move(in := 0, out1 => "UpDown".UD_0to1.V_BoxID_B)
   END_RUNG
   RUNG wire#w1
      "Enqueue3"("Array" := "CnvB".Sect0.V_ArrayBox, Input := "CnvB".Sect0.I_RFID_1, size := "CnvB".Sect0.V_NumOfBox)
   END_RUNG
   RUNG wire#w1
      Move(in := 0, out1 => "Boxes".Boxes["CnvB".Sect0.I_RFID_1].V_SectionOn)
   END_RUNG
   RUNG wire#w1
      Move(in := 1, out1 => "Boxes".Boxes["CnvB".Sect0.I_RFID_1].V_ConveyorOn)
   END_RUNG
   RUNG wire#w1
      Move(in := 1, out1 => "Boxes".Boxes["CnvB".Sect0.I_RFID_1].V_TypeOn)
   END_RUNG
   RUNG wire#w1
      Move(in := 2, out1 => "Boxes".Boxes["CnvB".Sect0.I_RFID_1].V_Direction)
   END_RUNG
   RUNG wire#w1
      R_Coil( "M_UD_0to1_B_7" )
   END_RUNG
   // the same network as SCL:
   #_w1 := "M_B_S0_1" AND ("CnvB".Sect0.I_RFID_1 > 0);
   #_w2 := #_w1 AND NOT "M_B_S0_1_Trig";   // rising edge
   "M_B_S0_1_Trig" := #_w1;
   IF #_w2 THEN
       "UpDown".UD_0to1.V_Busy_B := "UpDown".UD_0to1.V_Busy_B - 1;
       "UpDown".UD_0to1.V_BoxID_B := 0;
       "Enqueue3"("Array" := "CnvB".Sect0.V_ArrayBox,
                  Input := "CnvB".Sect0.I_RFID_1,
                  size := "CnvB".Sect0.V_NumOfBox);
       "Boxes".Boxes["CnvB".Sect0.I_RFID_1].V_SectionOn := 0;
       "Boxes".Boxes["CnvB".Sect0.I_RFID_1].V_ConveyorOn := 1;
       "Boxes".Boxes["CnvB".Sect0.I_RFID_1].V_TypeOn := 1;
       "Boxes".Boxes["CnvB".Sect0.I_RFID_1].V_Direction := 2;
       "M_UD_0to1_B_7" := FALSE;
   END_IF;
END_REGION

REGION Network 227: Mode back sect 0 output - activate
   RUNG wire#powerrail
      Contact( "M_B_S0_1" )
      { S7_Templates := "SrcType := DInt" } GT_Contact(in1 := "CnvB".Sect0.I_RFID_2, in2 := 0)
      S_Coil( "M_B_S0_2" )
   END_RUNG
   // the same network as SCL:
   IF "M_B_S0_1" AND ("CnvB".Sect0.I_RFID_2 > 0) THEN "M_B_S0_2" := TRUE; END_IF;
END_REGION

REGION Network 228: Mode back sect 0 output
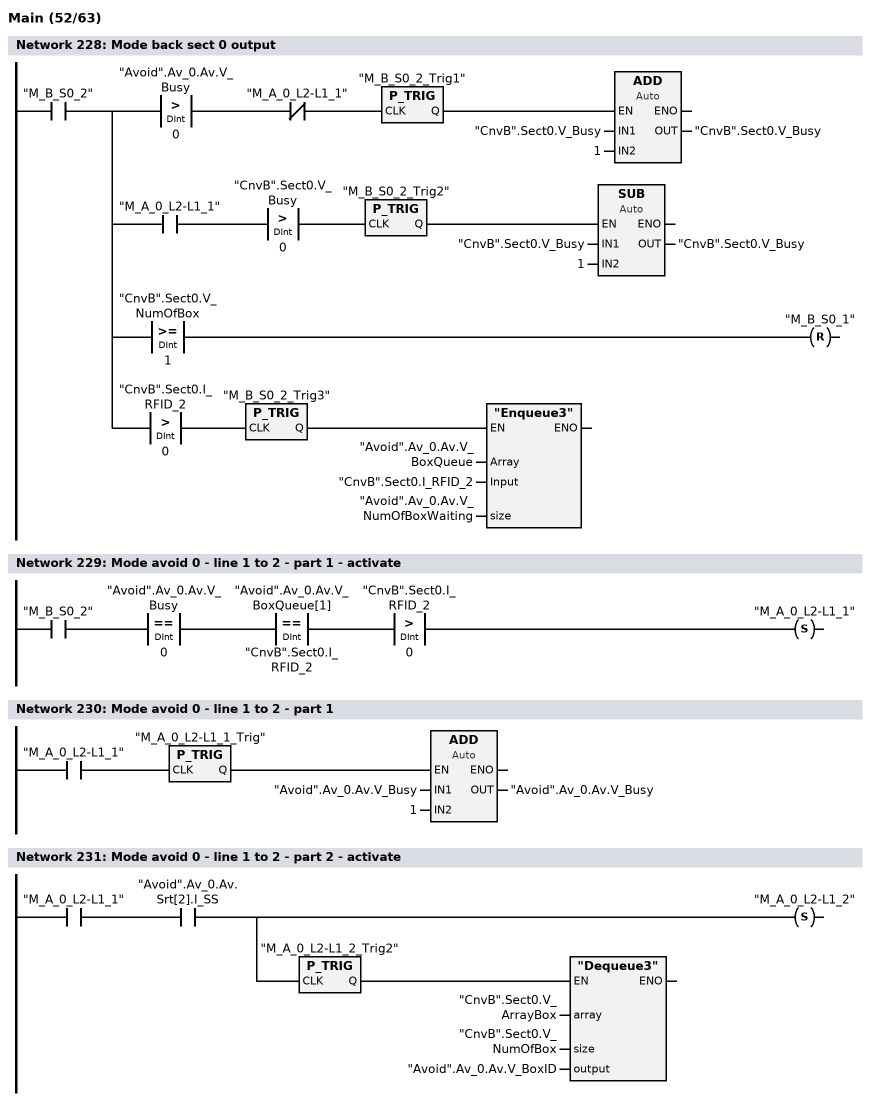
   RUNG wire#powerrail
      Contact( "M_B_S0_2" )
      wire#w1
      { S7_Templates := "SrcType := DInt" } GT_Contact(in1 := "Avoid".Av_0.Av.V_Busy, in2 := 0)
      I_Contact( "M_A_0_L2-L1_1" )
      P_Trig( "M_B_S0_2_Trig1" )
      Add(in1 := "CnvB".Sect0.V_Busy, in2 := 1, out => "CnvB".Sect0.V_Busy)
   END_RUNG
   RUNG wire#w1
      Contact( "M_A_0_L2-L1_1" )
      { S7_Templates := "SrcType := DInt" } GT_Contact(in1 := "CnvB".Sect0.V_Busy, in2 := 0)
      P_Trig( "M_B_S0_2_Trig2" )
      Sub(in1 := "CnvB".Sect0.V_Busy, in2 := 1, out => "CnvB".Sect0.V_Busy)
   END_RUNG
   RUNG wire#w1
      { S7_Templates := "SrcType := DInt" } GE_Contact(in1 := "CnvB".Sect0.V_NumOfBox, in2 := 1)
      R_Coil( "M_B_S0_1" )
   END_RUNG
   RUNG wire#w1
      { S7_Templates := "SrcType := DInt" } GT_Contact(in1 := "CnvB".Sect0.I_RFID_2, in2 := 0)
      P_Trig( "M_B_S0_2_Trig3" )
      "Enqueue3"("Array" := "Avoid".Av_0.Av.V_BoxQueue, Input := "CnvB".Sect0.I_RFID_2, size := "Avoid".Av_0.Av.V_NumOfBoxWaiting)
   END_RUNG
   // the same network as SCL:
   #_w1 := "M_B_S0_2" AND ("Avoid".Av_0.Av.V_Busy > 0) AND NOT "M_A_0_L2-L1_1";
   #_w2 := #_w1 AND NOT "M_B_S0_2_Trig1";   // rising edge
   "M_B_S0_2_Trig1" := #_w1;
   IF #_w2 THEN "CnvB".Sect0.V_Busy := "CnvB".Sect0.V_Busy + 1; END_IF;
   #_w3 := "M_B_S0_2" AND "M_A_0_L2-L1_1" AND ("CnvB".Sect0.V_Busy > 0);
   #_w4 := #_w3 AND NOT "M_B_S0_2_Trig2";   // rising edge
   "M_B_S0_2_Trig2" := #_w3;
   IF #_w4 THEN "CnvB".Sect0.V_Busy := "CnvB".Sect0.V_Busy - 1; END_IF;
   IF "M_B_S0_2" AND ("CnvB".Sect0.V_NumOfBox >= 1) THEN "M_B_S0_1" := FALSE; END_IF;
   #_w5 := "M_B_S0_2" AND ("CnvB".Sect0.I_RFID_2 > 0);
   #_w6 := #_w5 AND NOT "M_B_S0_2_Trig3";   // rising edge
   "M_B_S0_2_Trig3" := #_w5;
   IF #_w6 THEN
       "Enqueue3"("Array" := "Avoid".Av_0.Av.V_BoxQueue,
                  Input := "CnvB".Sect0.I_RFID_2,
                  size := "Avoid".Av_0.Av.V_NumOfBoxWaiting);
   END_IF;
END_REGION

REGION Network 229: Mode avoid 0 - line 1 to 2 - part 1 - activate
   RUNG wire#powerrail
      Contact( "M_B_S0_2" )
      { S7_Templates := "SrcType := DInt" } EQ_Contact(in1 := "Avoid".Av_0.Av.V_Busy, in2 := 0)
      { S7_Templates := "SrcType := DInt" } EQ_Contact(in1 := "Avoid".Av_0.Av.V_BoxQueue[1], in2 := "CnvB".Sect0.I_RFID_2)
      { S7_Templates := "SrcType := DInt" } GT_Contact(in1 := "CnvB".Sect0.I_RFID_2, in2 := 0)
      S_Coil( "M_A_0_L2-L1_1" )
   END_RUNG
   // the same network as SCL:
   IF "M_B_S0_2" AND ("Avoid".Av_0.Av.V_Busy = 0) AND ("Avoid".Av_0.Av.V_BoxQueue[1] = "CnvB".Sect0.I_RFID_2) AND ("CnvB".Sect0.I_RFID_2 > 0) THEN
       "M_A_0_L2-L1_1" := TRUE;
   END_IF;
END_REGION

REGION Network 230: Mode avoid 0 - line 1 to 2 - part 1
   RUNG wire#powerrail
      Contact( "M_A_0_L2-L1_1" )
      P_Trig( "M_A_0_L2-L1_1_Trig" )
      Add(in1 := "Avoid".Av_0.Av.V_Busy, in2 := 1, out => "Avoid".Av_0.Av.V_Busy)
   END_RUNG
   // the same network as SCL:
   #_w1 := "M_A_0_L2-L1_1" AND NOT "M_A_0_L2-L1_1_Trig";   // rising edge
   "M_A_0_L2-L1_1_Trig" := "M_A_0_L2-L1_1";
   IF #_w1 THEN "Avoid".Av_0.Av.V_Busy := "Avoid".Av_0.Av.V_Busy + 1; END_IF;
END_REGION

REGION Network 231: Mode avoid 0 - line 1 to 2 - part 2 - activate
   RUNG wire#powerrail
      Contact( "M_A_0_L2-L1_1" )
      Contact( "Avoid".Av_0.Av.Srt[2].I_SS )
      wire#w1
      S_Coil( "M_A_0_L2-L1_2" )
   END_RUNG
   RUNG wire#w1
      P_Trig( "M_A_0_L2-L1_2_Trig2" )
      "Dequeue3"("array" := "CnvB".Sect0.V_ArrayBox, size := "CnvB".Sect0.V_NumOfBox, output := "Avoid".Av_0.Av.V_BoxID)
   END_RUNG
   // the same network as SCL:
   #_w1 := "M_A_0_L2-L1_1" AND "Avoid".Av_0.Av.Srt[2].I_SS;
   IF #_w1 THEN "M_A_0_L2-L1_2" := TRUE; END_IF;
   #_w2 := #_w1 AND NOT "M_A_0_L2-L1_2_Trig2";   // rising edge
   "M_A_0_L2-L1_2_Trig2" := #_w1;
   IF #_w2 THEN
       "Dequeue3"("array" := "CnvB".Sect0.V_ArrayBox,
                  size := "CnvB".Sect0.V_NumOfBox,
                  output := "Avoid".Av_0.Av.V_BoxID);
   END_IF;
END_REGION

REGION Network 232: Mode avoid 0 - line 1 to 2 - part 2
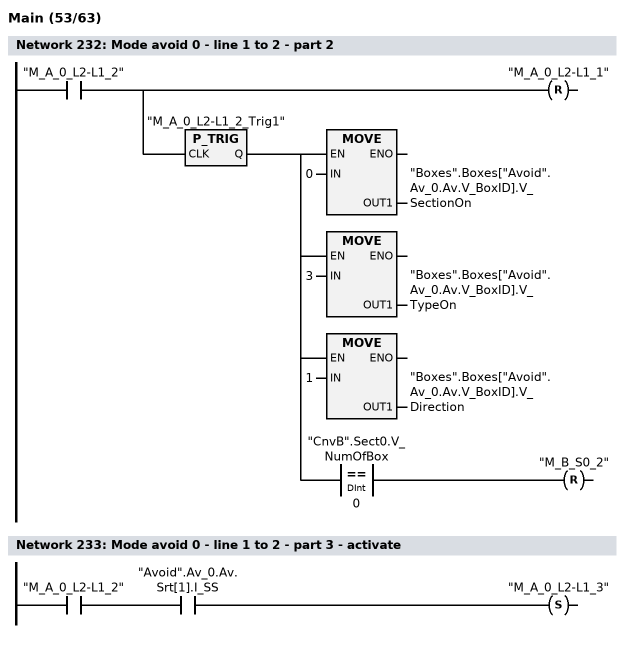
   RUNG wire#powerrail
      Contact( "M_A_0_L2-L1_2" )
      wire#w1
      R_Coil( "M_A_0_L2-L1_1" )
   END_RUNG
   RUNG wire#w1
      P_Trig( "M_A_0_L2-L1_2_Trig1" )
      wire#w2
      Move(in := 0, out1 => "Boxes".Boxes["Avoid".Av_0.Av.V_BoxID].V_SectionOn)
   END_RUNG
   RUNG wire#w2
      Move(in := 3, out1 => "Boxes".Boxes["Avoid".Av_0.Av.V_BoxID].V_TypeOn)
   END_RUNG
   RUNG wire#w2
      Move(in := 1, out1 => "Boxes".Boxes["Avoid".Av_0.Av.V_BoxID].V_Direction)
   END_RUNG
   RUNG wire#w2
      { S7_Templates := "SrcType := DInt" } EQ_Contact(in1 := "CnvB".Sect0.V_NumOfBox, in2 := 0)
      R_Coil( "M_B_S0_2" )
   END_RUNG
   // the same network as SCL:
   IF "M_A_0_L2-L1_2" THEN "M_A_0_L2-L1_1" := FALSE; END_IF;
   #_w1 := "M_A_0_L2-L1_2" AND NOT "M_A_0_L2-L1_2_Trig1";   // rising edge
   "M_A_0_L2-L1_2_Trig1" := "M_A_0_L2-L1_2";
   IF #_w1 THEN
       "Boxes".Boxes["Avoid".Av_0.Av.V_BoxID].V_SectionOn := 0;
       "Boxes".Boxes["Avoid".Av_0.Av.V_BoxID].V_TypeOn := 3;
       "Boxes".Boxes["Avoid".Av_0.Av.V_BoxID].V_Direction := 1;
   END_IF;
   IF #_w1 AND ("CnvB".Sect0.V_NumOfBox = 0) THEN "M_B_S0_2" := FALSE; END_IF;
END_REGION

REGION Network 233: Mode avoid 0 - line 1 to 2 - part 3 - activate
   RUNG wire#powerrail
      Contact( "M_A_0_L2-L1_2" )
      Contact( "Avoid".Av_0.Av.Srt[1].I_SS )
      S_Coil( "M_A_0_L2-L1_3" )
   END_RUNG
   // the same network as SCL:
   IF "M_A_0_L2-L1_2" AND "Avoid".Av_0.Av.Srt[1].I_SS THEN "M_A_0_L2-L1_3" := TRUE; END_IF;
END_REGION

REGION Network 234: Mode avoid 0 - line 1 to 2 - part 3
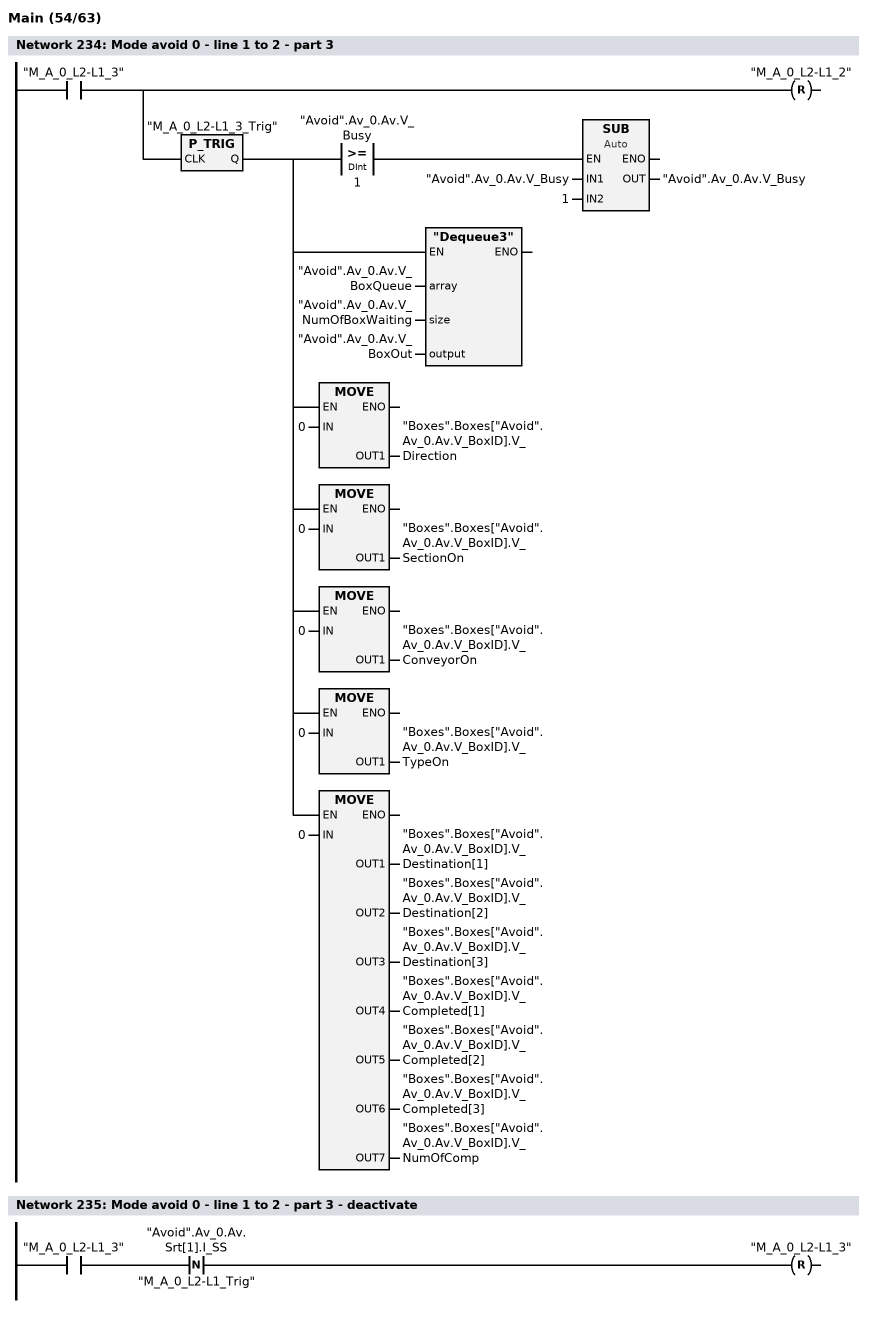
   RUNG wire#powerrail
      Contact( "M_A_0_L2-L1_3" )
      wire#w1
      R_Coil( "M_A_0_L2-L1_2" )
   END_RUNG
   RUNG wire#w1
      P_Trig( "M_A_0_L2-L1_3_Trig" )
      wire#w2
      { S7_Templates := "SrcType := DInt" } GE_Contact(in1 := "Avoid".Av_0.Av.V_Busy, in2 := 1)
      Sub(in1 := "Avoid".Av_0.Av.V_Busy, in2 := 1, out => "Avoid".Av_0.Av.V_Busy)
   END_RUNG
   RUNG wire#w2
      "Dequeue3"("array" := "Avoid".Av_0.Av.V_BoxQueue, size := "Avoid".Av_0.Av.V_NumOfBoxWaiting, output := "Avoid".Av_0.Av.V_BoxOut)
   END_RUNG
   RUNG wire#w2
      Move(in := 0, out1 => "Boxes".Boxes["Avoid".Av_0.Av.V_BoxID].V_Direction)
   END_RUNG
   RUNG wire#w2
      Move(in := 0, out1 => "Boxes".Boxes["Avoid".Av_0.Av.V_BoxID].V_SectionOn)
   END_RUNG
   RUNG wire#w2
      Move(in := 0, out1 => "Boxes".Boxes["Avoid".Av_0.Av.V_BoxID].V_ConveyorOn)
   END_RUNG
   RUNG wire#w2
      Move(in := 0, out1 => "Boxes".Boxes["Avoid".Av_0.Av.V_BoxID].V_TypeOn)
   END_RUNG
   RUNG wire#w2
      Move(in := 0, out1 => "Boxes".Boxes["Avoid".Av_0.Av.V_BoxID].V_Destination[1], out2 => "Boxes".Boxes["Avoid".Av_0.Av.V_BoxID].V_Destination[2], out3 => "Boxes".Boxes["Avoid".Av_0.Av.V_BoxID].V_Destination[3], out4 => "Boxes".Boxes["Avoid".Av_0.Av.V_BoxID].V_Completed[1], out5 => "Boxes".Boxes["Avoid".Av_0.Av.V_BoxID].V_Completed[2], out6 => "Boxes".Boxes["Avoid".Av_0.Av.V_BoxID].V_Completed[3], out7 => "Boxes".Boxes["Avoid".Av_0.Av.V_BoxID].V_NumOfComp)
   END_RUNG
   // the same network as SCL:
   IF "M_A_0_L2-L1_3" THEN "M_A_0_L2-L1_2" := FALSE; END_IF;
   #_w1 := "M_A_0_L2-L1_3" AND NOT "M_A_0_L2-L1_3_Trig";   // rising edge
   "M_A_0_L2-L1_3_Trig" := "M_A_0_L2-L1_3";
   IF #_w1 AND ("Avoid".Av_0.Av.V_Busy >= 1) THEN
       "Avoid".Av_0.Av.V_Busy := "Avoid".Av_0.Av.V_Busy - 1;
   END_IF;
   IF #_w1 THEN
       "Dequeue3"("array" := "Avoid".Av_0.Av.V_BoxQueue,
                  size := "Avoid".Av_0.Av.V_NumOfBoxWaiting,
                  output := "Avoid".Av_0.Av.V_BoxOut);
       "Boxes".Boxes["Avoid".Av_0.Av.V_BoxID].V_Direction := 0;
       "Boxes".Boxes["Avoid".Av_0.Av.V_BoxID].V_SectionOn := 0;
       "Boxes".Boxes["Avoid".Av_0.Av.V_BoxID].V_ConveyorOn := 0;
       "Boxes".Boxes["Avoid".Av_0.Av.V_BoxID].V_TypeOn := 0;
       "Boxes".Boxes["Avoid".Av_0.Av.V_BoxID].V_Destination[1] := 0;
       "Boxes".Boxes["Avoid".Av_0.Av.V_BoxID].V_Destination[2] := 0;
       "Boxes".Boxes["Avoid".Av_0.Av.V_BoxID].V_Destination[3] := 0;
       "Boxes".Boxes["Avoid".Av_0.Av.V_BoxID].V_Completed[1] := 0;
       "Boxes".Boxes["Avoid".Av_0.Av.V_BoxID].V_Completed[2] := 0;
       "Boxes".Boxes["Avoid".Av_0.Av.V_BoxID].V_Completed[3] := 0;
       "Boxes".Boxes["Avoid".Av_0.Av.V_BoxID].V_NumOfComp := 0;
   END_IF;
END_REGION

REGION Network 235: Mode avoid 0 - line 1 to 2 - part 3 - deactivate
   RUNG wire#powerrail
      Contact( "M_A_0_L2-L1_3" )
      N_Contact(operand := "Avoid".Av_0.Av.Srt[1].I_SS, bit := "M_A_0_L2-L1_Trig")
      R_Coil( "M_A_0_L2-L1_3" )
   END_RUNG
   // the same network as SCL:
   #_w1 := "M_A_0_L2-L1_3" AND NOT "Avoid".Av_0.Av.Srt[1].I_SS AND "M_A_0_L2-L1_Trig";   // falling edge of "Avoid".Av_0.Av.Srt[1].I_SS
   "M_A_0_L2-L1_Trig" := "Avoid".Av_0.Av.Srt[1].I_SS;
   IF #_w1 THEN "M_A_0_L2-L1_3" := FALSE; END_IF;
END_REGION

REGION Network 236: Motor Control - forward
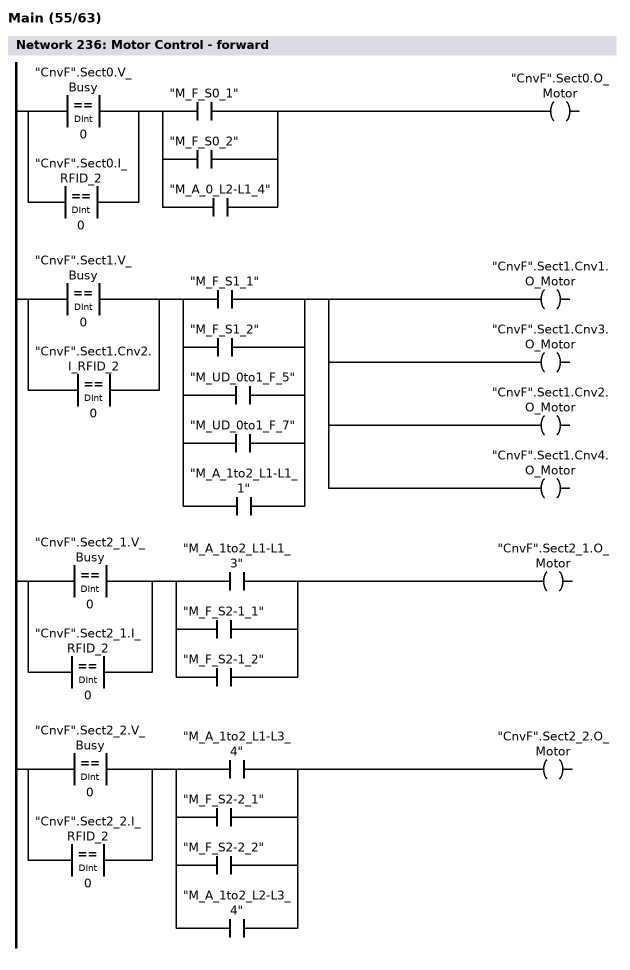
   RUNG wire#powerrail
      { S7_Templates := "SrcType := DInt" } EQ_Contact(in1 := "CnvF".Sect0.V_Busy, in2 := 0)
      wire#w1
      Contact( "M_F_S0_1" )
      wire#w2
      Coil( "CnvF".Sect0.O_Motor )
   END_RUNG
   RUNG wire#powerrail
      { S7_Templates := "SrcType := DInt" } EQ_Contact(in1 := "CnvF".Sect0.I_RFID_2, in2 := 0)
   END_RUNG wire#w1
   RUNG wire#w1
      Contact( "M_F_S0_2" )
   END_RUNG wire#w2
   RUNG wire#w1
      Contact( "M_A_0_L2-L1_4" )
   END_RUNG wire#w2
   RUNG wire#powerrail
      { S7_Templates := "SrcType := DInt" } EQ_Contact(in1 := "CnvF".Sect1.V_Busy, in2 := 0)
      wire#w3
      Contact( "M_F_S1_1" )
      wire#w4
      Coil( "CnvF".Sect1.Cnv1.O_Motor )
   END_RUNG
   RUNG wire#powerrail
      { S7_Templates := "SrcType := DInt" } EQ_Contact(in1 := "CnvF".Sect1.Cnv2.I_RFID_2, in2 := 0)
   END_RUNG wire#w3
   RUNG wire#w3
      Contact( "M_F_S1_2" )
   END_RUNG wire#w4
   RUNG wire#w3
      Contact( "M_UD_0to1_F_5" )
   END_RUNG wire#w4
   RUNG wire#w3
      Contact( "M_UD_0to1_F_7" )
   END_RUNG wire#w4
   RUNG wire#w3
      Contact( "M_A_1to2_L1-L1_1" )
   END_RUNG wire#w4
   RUNG wire#w4
      Coil( "CnvF".Sect1.Cnv3.O_Motor )
   END_RUNG
   RUNG wire#w4
      Coil( "CnvF".Sect1.Cnv2.O_Motor )
   END_RUNG
   RUNG wire#w4
      Coil( "CnvF".Sect1.Cnv4.O_Motor )
   END_RUNG
   RUNG wire#powerrail
      { S7_Templates := "SrcType := DInt" } EQ_Contact(in1 := "CnvF".Sect2_1.V_Busy, in2 := 0)
      wire#w5
      Contact( "M_A_1to2_L1-L1_3" )
      wire#w6
      Coil( "CnvF".Sect2_1.O_Motor )
   END_RUNG
   RUNG wire#powerrail
      { S7_Templates := "SrcType := DInt" } EQ_Contact(in1 := "CnvF".Sect2_1.I_RFID_2, in2 := 0)
   END_RUNG wire#w5
   RUNG wire#w5
      Contact( "M_F_S2-1_1" )
   END_RUNG wire#w6
   RUNG wire#w5
      Contact( "M_F_S2-1_2" )
   END_RUNG wire#w6
   RUNG wire#powerrail
      { S7_Templates := "SrcType := DInt" } EQ_Contact(in1 := "CnvF".Sect2_2.V_Busy, in2 := 0)
      wire#w7
      Contact( "M_A_1to2_L1-L3_4" )
      wire#w8
      Coil( "CnvF".Sect2_2.O_Motor )
   END_RUNG
   RUNG wire#powerrail
      { S7_Templates := "SrcType := DInt" } EQ_Contact(in1 := "CnvF".Sect2_2.I_RFID_2, in2 := 0)
   END_RUNG wire#w7
   RUNG wire#w7
      Contact( "M_F_S2-2_1" )
   END_RUNG wire#w8
   RUNG wire#w7
      Contact( "M_F_S2-2_2" )
   END_RUNG wire#w8
   RUNG wire#w7
      Contact( "M_A_1to2_L2-L3_4" )
   END_RUNG wire#w8
   // the same network as SCL:
   "CnvF".Sect0.O_Motor := (("CnvF".Sect0.V_Busy = 0) OR ("CnvF".Sect0.I_RFID_2 = 0)) AND ("M_F_S0_1" OR "M_F_S0_2" OR "M_A_0_L2-L1_4");
   "CnvF".Sect1.Cnv1.O_Motor := (("CnvF".Sect1.V_Busy = 0) OR ("CnvF".Sect1.Cnv2.I_RFID_2 = 0)) AND ("M_F_S1_1" OR "M_F_S1_2" OR "M_UD_0to1_F_5" OR "M_UD_0to1_F_7" OR "M_A_1to2_L1-L1_1");
   "CnvF".Sect1.Cnv3.O_Motor := "CnvF".Sect1.Cnv1.O_Motor;
   "CnvF".Sect1.Cnv2.O_Motor := "CnvF".Sect1.Cnv1.O_Motor;
   "CnvF".Sect1.Cnv4.O_Motor := "CnvF".Sect1.Cnv1.O_Motor;
   "CnvF".Sect2_1.O_Motor := (("CnvF".Sect2_1.V_Busy = 0) OR ("CnvF".Sect2_1.I_RFID_2 = 0)) AND ("M_A_1to2_L1-L1_3" OR "M_F_S2-1_1" OR "M_F_S2-1_2");
   "CnvF".Sect2_2.O_Motor := (("CnvF".Sect2_2.V_Busy = 0) OR ("CnvF".Sect2_2.I_RFID_2 = 0)) AND ("M_A_1to2_L1-L3_4" OR "M_F_S2-2_1" OR "M_F_S2-2_2" OR "M_A_1to2_L2-L3_4");
END_REGION

REGION Network 237: Motor Control - back
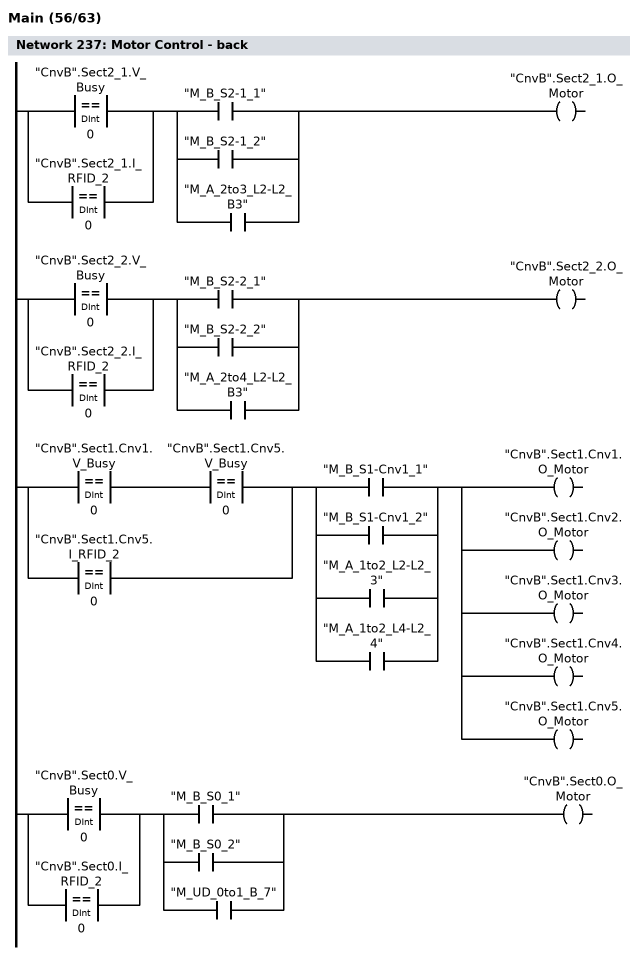
   RUNG wire#powerrail
      { S7_Templates := "SrcType := DInt" } EQ_Contact(in1 := "CnvB".Sect2_1.V_Busy, in2 := 0)
      wire#w1
      Contact( "M_B_S2-1_1" )
      wire#w2
      Coil( "CnvB".Sect2_1.O_Motor )
   END_RUNG
   RUNG wire#powerrail
      { S7_Templates := "SrcType := DInt" } EQ_Contact(in1 := "CnvB".Sect2_1.I_RFID_2, in2 := 0)
   END_RUNG wire#w1
   RUNG wire#w1
      Contact( "M_B_S2-1_2" )
   END_RUNG wire#w2
   RUNG wire#w1
      Contact( "M_A_2to3_L2-L2_B3" )
   END_RUNG wire#w2
   RUNG wire#powerrail
      { S7_Templates := "SrcType := DInt" } EQ_Contact(in1 := "CnvB".Sect2_2.V_Busy, in2 := 0)
      wire#w3
      Contact( "M_B_S2-2_1" )
      wire#w4
      Coil( "CnvB".Sect2_2.O_Motor )
   END_RUNG
   RUNG wire#powerrail
      { S7_Templates := "SrcType := DInt" } EQ_Contact(in1 := "CnvB".Sect2_2.I_RFID_2, in2 := 0)
   END_RUNG wire#w3
   RUNG wire#w3
      Contact( "M_B_S2-2_2" )
   END_RUNG wire#w4
   RUNG wire#w3
      Contact( "M_A_2to4_L2-L2_B3" )
   END_RUNG wire#w4
   RUNG wire#powerrail
      { S7_Templates := "SrcType := DInt" } EQ_Contact(in1 := "CnvB".Sect1.Cnv1.V_Busy, in2 := 0)
      { S7_Templates := "SrcType := DInt" } EQ_Contact(in1 := "CnvB".Sect1.Cnv5.V_Busy, in2 := 0)
      wire#w5
      Contact( "M_B_S1-Cnv1_1" )
      wire#w6
      Coil( "CnvB".Sect1.Cnv1.O_Motor )
   END_RUNG
   RUNG wire#powerrail
      { S7_Templates := "SrcType := DInt" } EQ_Contact(in1 := "CnvB".Sect1.Cnv5.I_RFID_2, in2 := 0)
   END_RUNG wire#w5
   RUNG wire#w5
      Contact( "M_B_S1-Cnv1_2" )
   END_RUNG wire#w6
   RUNG wire#w5
      Contact( "M_A_1to2_L2-L2_3" )
   END_RUNG wire#w6
   RUNG wire#w5
      Contact( "M_A_1to2_L4-L2_4" )
   END_RUNG wire#w6
   RUNG wire#w6
      Coil( "CnvB".Sect1.Cnv2.O_Motor )
   END_RUNG
   RUNG wire#w6
      Coil( "CnvB".Sect1.Cnv3.O_Motor )
   END_RUNG
   RUNG wire#w6
      Coil( "CnvB".Sect1.Cnv4.O_Motor )
   END_RUNG
   RUNG wire#w6
      Coil( "CnvB".Sect1.Cnv5.O_Motor )
   END_RUNG
   RUNG wire#powerrail
      { S7_Templates := "SrcType := DInt" } EQ_Contact(in1 := "CnvB".Sect0.V_Busy, in2 := 0)
      wire#w7
      Contact( "M_B_S0_1" )
      wire#w8
      Coil( "CnvB".Sect0.O_Motor )
   END_RUNG
   RUNG wire#powerrail
      { S7_Templates := "SrcType := DInt" } EQ_Contact(in1 := "CnvB".Sect0.I_RFID_2, in2 := 0)
   END_RUNG wire#w7
   RUNG wire#w7
      Contact( "M_B_S0_2" )
   END_RUNG wire#w8
   RUNG wire#w7
      Contact( "M_UD_0to1_B_7" )
   END_RUNG wire#w8
   // the same network as SCL:
   "CnvB".Sect2_1.O_Motor := (("CnvB".Sect2_1.V_Busy = 0) OR ("CnvB".Sect2_1.I_RFID_2 = 0)) AND ("M_B_S2-1_1" OR "M_B_S2-1_2" OR "M_A_2to3_L2-L2_B3");
   "CnvB".Sect2_2.O_Motor := (("CnvB".Sect2_2.V_Busy = 0) OR ("CnvB".Sect2_2.I_RFID_2 = 0)) AND ("M_B_S2-2_1" OR "M_B_S2-2_2" OR "M_A_2to4_L2-L2_B3");
   "CnvB".Sect1.Cnv1.O_Motor := ((("CnvB".Sect1.Cnv1.V_Busy = 0) AND ("CnvB".Sect1.Cnv5.V_Busy = 0)) OR ("CnvB".Sect1.Cnv5.I_RFID_2 = 0)) AND ("M_B_S1-Cnv1_1" OR "M_B_S1-Cnv1_2" OR "M_A_1to2_L2-L2_3" OR "M_A_1to2_L4-L2_4");
   "CnvB".Sect1.Cnv2.O_Motor := "CnvB".Sect1.Cnv1.O_Motor;
   "CnvB".Sect1.Cnv3.O_Motor := "CnvB".Sect1.Cnv1.O_Motor;
   "CnvB".Sect1.Cnv4.O_Motor := "CnvB".Sect1.Cnv1.O_Motor;
   "CnvB".Sect1.Cnv5.O_Motor := "CnvB".Sect1.Cnv1.O_Motor;
   "CnvB".Sect0.O_Motor := (("CnvB".Sect0.V_Busy = 0) OR ("CnvB".Sect0.I_RFID_2 = 0)) AND ("M_B_S0_1" OR "M_B_S0_2" OR "M_UD_0to1_B_7");
END_REGION

REGION Network 238: Motor Control - 2d frw
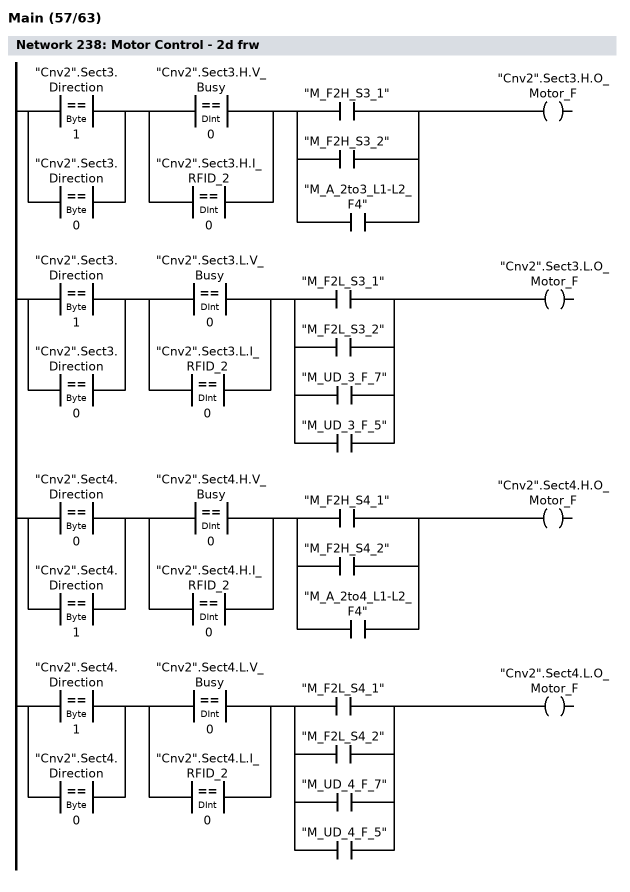
   RUNG wire#powerrail
      { S7_Templates := "SrcType := Byte" } EQ_Contact(in1 := "Cnv2".Sect3.Direction, in2 := 1)
      wire#w1
      { S7_Templates := "SrcType := DInt" } EQ_Contact(in1 := "Cnv2".Sect3.H.V_Busy, in2 := 0)
      wire#w2
      Contact( "M_F2H_S3_1" )
      wire#w3
      Coil( "Cnv2".Sect3.H.O_Motor_F )
   END_RUNG
   RUNG wire#powerrail
      { S7_Templates := "SrcType := Byte" } EQ_Contact(in1 := "Cnv2".Sect3.Direction, in2 := 0)
   END_RUNG wire#w1
   RUNG wire#w1
      { S7_Templates := "SrcType := DInt" } EQ_Contact(in1 := "Cnv2".Sect3.H.I_RFID_2, in2 := 0)
   END_RUNG wire#w2
   RUNG wire#w2
      Contact( "M_F2H_S3_2" )
   END_RUNG wire#w3
   RUNG wire#w2
      Contact( "M_A_2to3_L1-L2_F4" )
   END_RUNG wire#w3
   RUNG wire#powerrail
      { S7_Templates := "SrcType := Byte" } EQ_Contact(in1 := "Cnv2".Sect3.Direction, in2 := 1)
      wire#w4
      { S7_Templates := "SrcType := DInt" } EQ_Contact(in1 := "Cnv2".Sect3.L.V_Busy, in2 := 0)
      wire#w5
      Contact( "M_F2L_S3_1" )
      wire#w6
      Coil( "Cnv2".Sect3.L.O_Motor_F )
   END_RUNG
   RUNG wire#powerrail
      { S7_Templates := "SrcType := Byte" } EQ_Contact(in1 := "Cnv2".Sect3.Direction, in2 := 0)
   END_RUNG wire#w4
   RUNG wire#w4
      { S7_Templates := "SrcType := DInt" } EQ_Contact(in1 := "Cnv2".Sect3.L.I_RFID_2, in2 := 0)
   END_RUNG wire#w5
   RUNG wire#w5
      Contact( "M_F2L_S3_2" )
   END_RUNG wire#w6
   RUNG wire#w5
      Contact( "M_UD_3_F_7" )
   END_RUNG wire#w6
   RUNG wire#w5
      Contact( "M_UD_3_F_5" )
   END_RUNG wire#w6
   RUNG wire#powerrail
      { S7_Templates := "SrcType := Byte" } EQ_Contact(in1 := "Cnv2".Sect4.Direction, in2 := 0)
      wire#w7
      { S7_Templates := "SrcType := DInt" } EQ_Contact(in1 := "Cnv2".Sect4.H.V_Busy, in2 := 0)
      wire#w8
      Contact( "M_F2H_S4_1" )
      wire#w9
      Coil( "Cnv2".Sect4.H.O_Motor_F )
   END_RUNG
   RUNG wire#powerrail
      { S7_Templates := "SrcType := Byte" } EQ_Contact(in1 := "Cnv2".Sect4.Direction, in2 := 1)
   END_RUNG wire#w7
   RUNG wire#w7
      { S7_Templates := "SrcType := DInt" } EQ_Contact(in1 := "Cnv2".Sect4.H.I_RFID_2, in2 := 0)
   END_RUNG wire#w8
   RUNG wire#w8
      Contact( "M_F2H_S4_2" )
   END_RUNG wire#w9
   RUNG wire#w8
      Contact( "M_A_2to4_L1-L2_F4" )
   END_RUNG wire#w9
   RUNG wire#powerrail
      { S7_Templates := "SrcType := Byte" } EQ_Contact(in1 := "Cnv2".Sect4.Direction, in2 := 1)
      wire#w10
      { S7_Templates := "SrcType := DInt" } EQ_Contact(in1 := "Cnv2".Sect4.L.V_Busy, in2 := 0)
      wire#w11
      Contact( "M_F2L_S4_1" )
      wire#w12
      Coil( "Cnv2".Sect4.L.O_Motor_F )
   END_RUNG
   RUNG wire#powerrail
      { S7_Templates := "SrcType := Byte" } EQ_Contact(in1 := "Cnv2".Sect4.Direction, in2 := 0)
   END_RUNG wire#w10
   RUNG wire#w10
      { S7_Templates := "SrcType := DInt" } EQ_Contact(in1 := "Cnv2".Sect4.L.I_RFID_2, in2 := 0)
   END_RUNG wire#w11
   RUNG wire#w11
      Contact( "M_F2L_S4_2" )
   END_RUNG wire#w12
   RUNG wire#w11
      Contact( "M_UD_4_F_7" )
   END_RUNG wire#w12
   RUNG wire#w11
      Contact( "M_UD_4_F_5" )
   END_RUNG wire#w12
   // the same network as SCL:
   "Cnv2".Sect3.H.O_Motor_F := (("Cnv2".Sect3.Direction = 1) OR ("Cnv2".Sect3.Direction = 0)) AND (("Cnv2".Sect3.H.V_Busy = 0) OR ("Cnv2".Sect3.H.I_RFID_2 = 0)) AND ("M_F2H_S3_1" OR "M_F2H_S3_2" OR "M_A_2to3_L1-L2_F4");
   "Cnv2".Sect3.L.O_Motor_F := (("Cnv2".Sect3.Direction = 1) OR ("Cnv2".Sect3.Direction = 0)) AND (("Cnv2".Sect3.L.V_Busy = 0) OR ("Cnv2".Sect3.L.I_RFID_2 = 0)) AND ("M_F2L_S3_1" OR "M_F2L_S3_2" OR "M_UD_3_F_7" OR "M_UD_3_F_5");
   "Cnv2".Sect4.H.O_Motor_F := (("Cnv2".Sect4.Direction = 0) OR ("Cnv2".Sect4.Direction = 1)) AND (("Cnv2".Sect4.H.V_Busy = 0) OR ("Cnv2".Sect4.H.I_RFID_2 = 0)) AND ("M_F2H_S4_1" OR "M_F2H_S4_2" OR "M_A_2to4_L1-L2_F4");
   "Cnv2".Sect4.L.O_Motor_F := (("Cnv2".Sect4.Direction = 1) OR ("Cnv2".Sect4.Direction = 0)) AND (("Cnv2".Sect4.L.V_Busy = 0) OR ("Cnv2".Sect4.L.I_RFID_2 = 0)) AND ("M_F2L_S4_1" OR "M_F2L_S4_2" OR "M_UD_4_F_7" OR "M_UD_4_F_5");
END_REGION

REGION Network 239: Motor control - 2d back
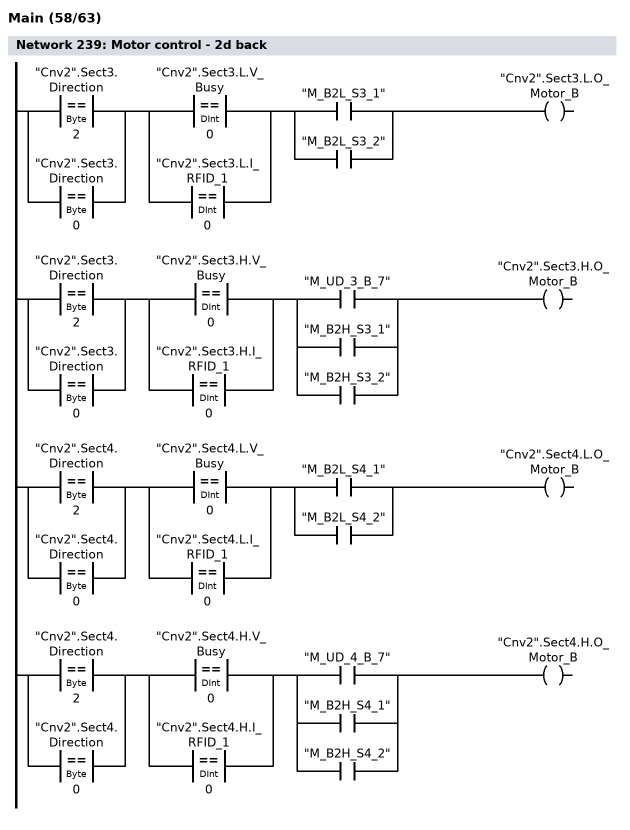
   RUNG wire#powerrail
      { S7_Templates := "SrcType := Byte" } EQ_Contact(in1 := "Cnv2".Sect3.Direction, in2 := 2)
      wire#w1
      { S7_Templates := "SrcType := DInt" } EQ_Contact(in1 := "Cnv2".Sect3.L.V_Busy, in2 := 0)
      wire#w2
      Contact( "M_B2L_S3_1" )
      wire#w3
      Coil( "Cnv2".Sect3.L.O_Motor_B )
   END_RUNG
   RUNG wire#powerrail
      { S7_Templates := "SrcType := Byte" } EQ_Contact(in1 := "Cnv2".Sect3.Direction, in2 := 0)
   END_RUNG wire#w1
   RUNG wire#w1
      { S7_Templates := "SrcType := DInt" } EQ_Contact(in1 := "Cnv2".Sect3.L.I_RFID_1, in2 := 0)
   END_RUNG wire#w2
   RUNG wire#w2
      Contact( "M_B2L_S3_2" )
   END_RUNG wire#w3
   RUNG wire#powerrail
      { S7_Templates := "SrcType := Byte" } EQ_Contact(in1 := "Cnv2".Sect3.Direction, in2 := 2)
      wire#w4
      { S7_Templates := "SrcType := DInt" } EQ_Contact(in1 := "Cnv2".Sect3.H.V_Busy, in2 := 0)
      wire#w5
      Contact( "M_UD_3_B_7" )
      wire#w6
      Coil( "Cnv2".Sect3.H.O_Motor_B )
   END_RUNG
   RUNG wire#powerrail
      { S7_Templates := "SrcType := Byte" } EQ_Contact(in1 := "Cnv2".Sect3.Direction, in2 := 0)
   END_RUNG wire#w4
   RUNG wire#w4
      { S7_Templates := "SrcType := DInt" } EQ_Contact(in1 := "Cnv2".Sect3.H.I_RFID_1, in2 := 0)
   END_RUNG wire#w5
   RUNG wire#w5
      Contact( "M_B2H_S3_1" )
   END_RUNG wire#w6
   RUNG wire#w5
      Contact( "M_B2H_S3_2" )
   END_RUNG wire#w6
   RUNG wire#powerrail
      { S7_Templates := "SrcType := Byte" } EQ_Contact(in1 := "Cnv2".Sect4.Direction, in2 := 2)
      wire#w7
      { S7_Templates := "SrcType := DInt" } EQ_Contact(in1 := "Cnv2".Sect4.L.V_Busy, in2 := 0)
      wire#w8
      Contact( "M_B2L_S4_1" )
      wire#w9
      Coil( "Cnv2".Sect4.L.O_Motor_B )
   END_RUNG
   RUNG wire#powerrail
      { S7_Templates := "SrcType := Byte" } EQ_Contact(in1 := "Cnv2".Sect4.Direction, in2 := 0)
   END_RUNG wire#w7
   RUNG wire#w7
      { S7_Templates := "SrcType := DInt" } EQ_Contact(in1 := "Cnv2".Sect4.L.I_RFID_1, in2 := 0)
   END_RUNG wire#w8
   RUNG wire#w8
      Contact( "M_B2L_S4_2" )
   END_RUNG wire#w9
   RUNG wire#powerrail
      { S7_Templates := "SrcType := Byte" } EQ_Contact(in1 := "Cnv2".Sect4.Direction, in2 := 2)
      wire#w10
      { S7_Templates := "SrcType := DInt" } EQ_Contact(in1 := "Cnv2".Sect4.H.V_Busy, in2 := 0)
      wire#w11
      Contact( "M_UD_4_B_7" )
      wire#w12
      Coil( "Cnv2".Sect4.H.O_Motor_B )
   END_RUNG
   RUNG wire#powerrail
      { S7_Templates := "SrcType := Byte" } EQ_Contact(in1 := "Cnv2".Sect4.Direction, in2 := 0)
   END_RUNG wire#w10
   RUNG wire#w10
      { S7_Templates := "SrcType := DInt" } EQ_Contact(in1 := "Cnv2".Sect4.H.I_RFID_1, in2 := 0)
   END_RUNG wire#w11
   RUNG wire#w11
      Contact( "M_B2H_S4_1" )
   END_RUNG wire#w12
   RUNG wire#w11
      Contact( "M_B2H_S4_2" )
   END_RUNG wire#w12
   // the same network as SCL:
   "Cnv2".Sect3.L.O_Motor_B := (("Cnv2".Sect3.Direction = 2) OR ("Cnv2".Sect3.Direction = 0)) AND (("Cnv2".Sect3.L.V_Busy = 0) OR ("Cnv2".Sect3.L.I_RFID_1 = 0)) AND ("M_B2L_S3_1" OR "M_B2L_S3_2");
   "Cnv2".Sect3.H.O_Motor_B := (("Cnv2".Sect3.Direction = 2) OR ("Cnv2".Sect3.Direction = 0)) AND (("Cnv2".Sect3.H.V_Busy = 0) OR ("Cnv2".Sect3.H.I_RFID_1 = 0)) AND ("M_UD_3_B_7" OR "M_B2H_S3_1" OR "M_B2H_S3_2");
   "Cnv2".Sect4.L.O_Motor_B := (("Cnv2".Sect4.Direction = 2) OR ("Cnv2".Sect4.Direction = 0)) AND (("Cnv2".Sect4.L.V_Busy = 0) OR ("Cnv2".Sect4.L.I_RFID_1 = 0)) AND ("M_B2L_S4_1" OR "M_B2L_S4_2");
   "Cnv2".Sect4.H.O_Motor_B := (("Cnv2".Sect4.Direction = 2) OR ("Cnv2".Sect4.Direction = 0)) AND (("Cnv2".Sect4.H.V_Busy = 0) OR ("Cnv2".Sect4.H.I_RFID_1 = 0)) AND ("M_UD_4_B_7" OR "M_B2H_S4_1" OR "M_B2H_S4_2");
END_REGION

REGION Network 240: Motor Control - updown 1to2
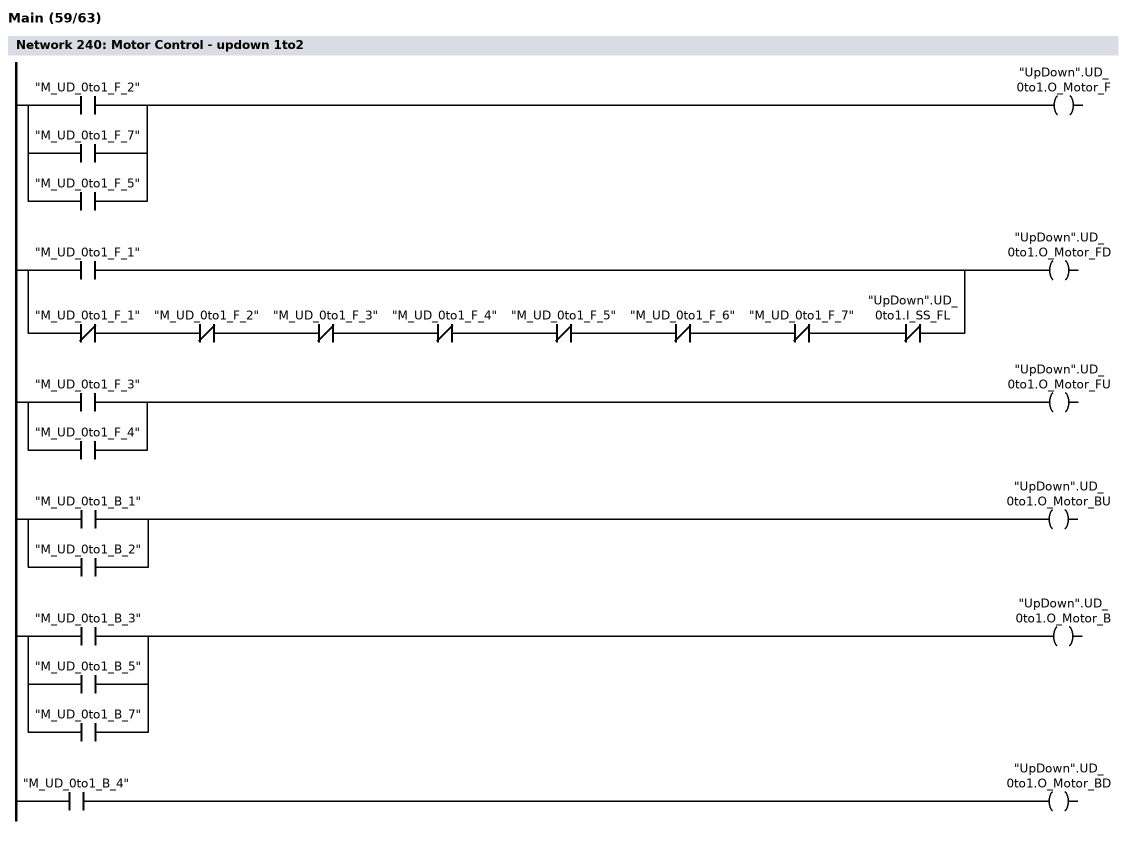
   RUNG wire#powerrail
      Contact( "M_UD_0to1_F_2" )
      wire#w1
      Coil( "UpDown".UD_0to1.O_Motor_F )
   END_RUNG
   RUNG wire#powerrail
      Contact( "M_UD_0to1_F_7" )
   END_RUNG wire#w1
   RUNG wire#powerrail
      Contact( "M_UD_0to1_F_5" )
   END_RUNG wire#w1
   RUNG wire#powerrail
      Contact( "M_UD_0to1_F_1" )
      wire#w2
      Coil( "UpDown".UD_0to1.O_Motor_FD )
   END_RUNG
   RUNG wire#powerrail
      I_Contact( "M_UD_0to1_F_1" )
      I_Contact( "M_UD_0to1_F_2" )
      I_Contact( "M_UD_0to1_F_3" )
      I_Contact( "M_UD_0to1_F_4" )
      I_Contact( "M_UD_0to1_F_5" )
      I_Contact( "M_UD_0to1_F_6" )
      I_Contact( "M_UD_0to1_F_7" )
      I_Contact( "UpDown".UD_0to1.I_SS_FL )
   END_RUNG wire#w2
   RUNG wire#powerrail
      Contact( "M_UD_0to1_F_3" )
      wire#w3
      Coil( "UpDown".UD_0to1.O_Motor_FU )
   END_RUNG
   RUNG wire#powerrail
      Contact( "M_UD_0to1_F_4" )
   END_RUNG wire#w3
   RUNG wire#powerrail
      Contact( "M_UD_0to1_B_1" )
      wire#w4
      Coil( "UpDown".UD_0to1.O_Motor_BU )
   END_RUNG
   RUNG wire#powerrail
      Contact( "M_UD_0to1_B_2" )
   END_RUNG wire#w4
   RUNG wire#powerrail
      Contact( "M_UD_0to1_B_3" )
      wire#w5
      Coil( "UpDown".UD_0to1.O_Motor_B )
   END_RUNG
   RUNG wire#powerrail
      Contact( "M_UD_0to1_B_5" )
   END_RUNG wire#w5
   RUNG wire#powerrail
      Contact( "M_UD_0to1_B_7" )
   END_RUNG wire#w5
   RUNG wire#powerrail
      Contact( "M_UD_0to1_B_4" )
      Coil( "UpDown".UD_0to1.O_Motor_BD )
   END_RUNG
   // the same network as SCL:
   "UpDown".UD_0to1.O_Motor_F := "M_UD_0to1_F_2" OR "M_UD_0to1_F_7" OR "M_UD_0to1_F_5";
   "UpDown".UD_0to1.O_Motor_FD := "M_UD_0to1_F_1" OR (NOT "M_UD_0to1_F_1" AND NOT "M_UD_0to1_F_2" AND NOT "M_UD_0to1_F_3" AND NOT "M_UD_0to1_F_4" AND NOT "M_UD_0to1_F_5" AND NOT "M_UD_0to1_F_6" AND NOT "M_UD_0to1_F_7" AND NOT "UpDown".UD_0to1.I_SS_FL);
   "UpDown".UD_0to1.O_Motor_FU := "M_UD_0to1_F_3" OR "M_UD_0to1_F_4";
   "UpDown".UD_0to1.O_Motor_BU := "M_UD_0to1_B_1" OR "M_UD_0to1_B_2";
   "UpDown".UD_0to1.O_Motor_B := "M_UD_0to1_B_3" OR "M_UD_0to1_B_5" OR "M_UD_0to1_B_7";
   "UpDown".UD_0to1.O_Motor_BD := "M_UD_0to1_B_4";
END_REGION

REGION Network 241: Motor Control - updown 3
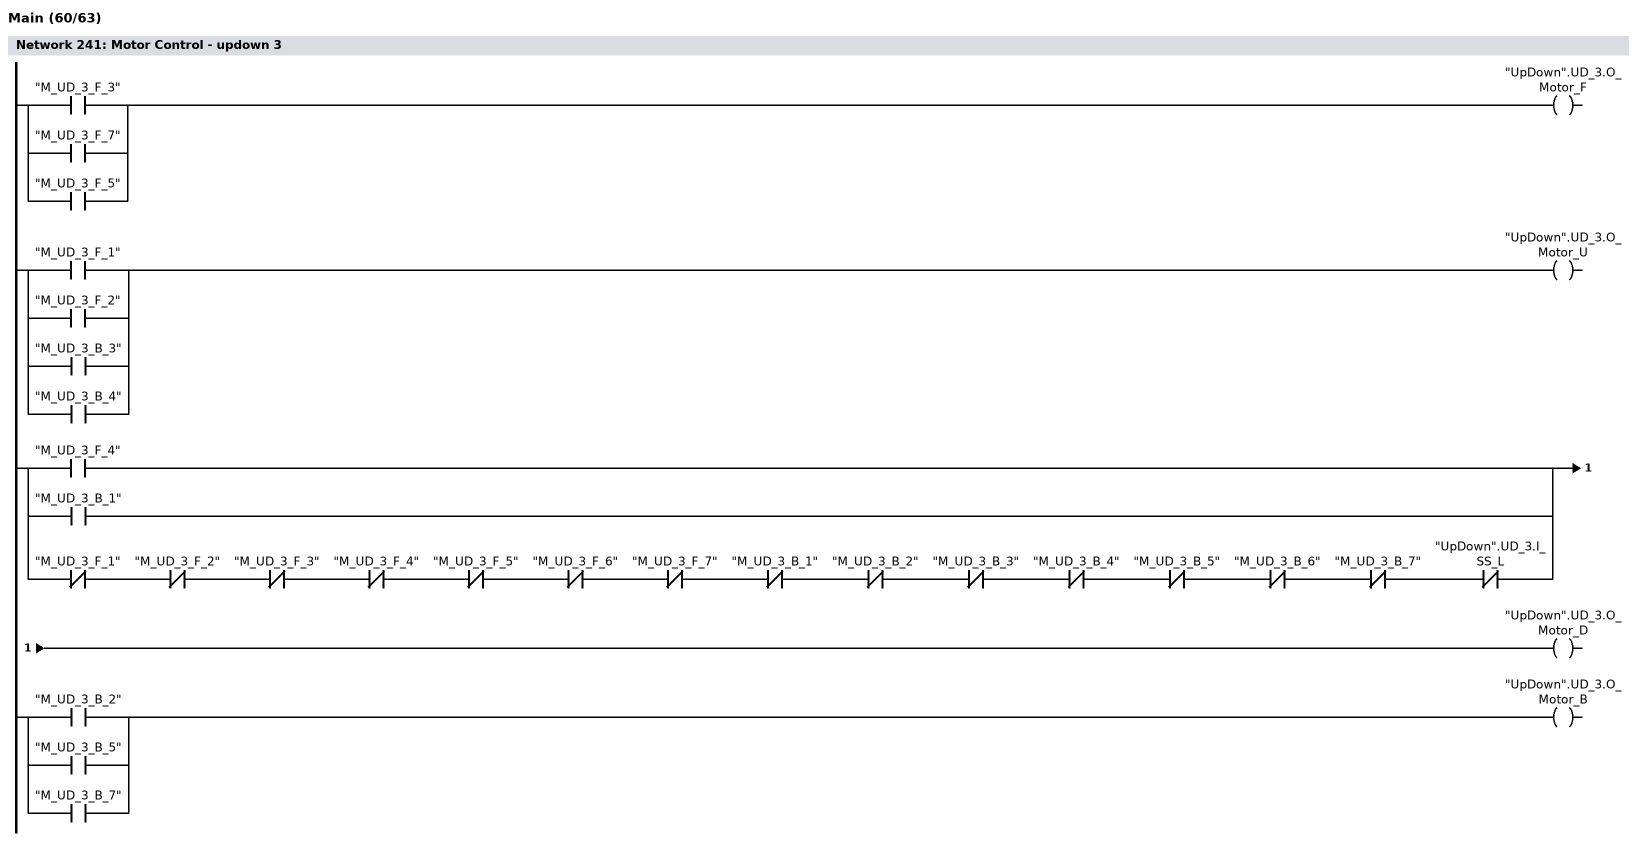
   RUNG wire#powerrail
      Contact( "M_UD_3_F_3" )
      wire#w1
      Coil( "UpDown".UD_3.O_Motor_F )
   END_RUNG
   RUNG wire#powerrail
      Contact( "M_UD_3_F_7" )
   END_RUNG wire#w1
   RUNG wire#powerrail
      Contact( "M_UD_3_F_5" )
   END_RUNG wire#w1
   RUNG wire#powerrail
      Contact( "M_UD_3_F_1" )
      wire#w2
      Coil( "UpDown".UD_3.O_Motor_U )
   END_RUNG
   RUNG wire#powerrail
      Contact( "M_UD_3_F_2" )
   END_RUNG wire#w2
   RUNG wire#powerrail
      Contact( "M_UD_3_B_3" )
   END_RUNG wire#w2
   RUNG wire#powerrail
      Contact( "M_UD_3_B_4" )
   END_RUNG wire#w2
   RUNG wire#powerrail
      Contact( "M_UD_3_F_4" )
      wire#w3
      Coil( "UpDown".UD_3.O_Motor_D )
   END_RUNG
   RUNG wire#powerrail
      Contact( "M_UD_3_B_1" )
   END_RUNG wire#w3
   RUNG wire#powerrail
      I_Contact( "M_UD_3_F_1" )
      I_Contact( "M_UD_3_F_2" )
      I_Contact( "M_UD_3_F_3" )
      I_Contact( "M_UD_3_F_4" )
      I_Contact( "M_UD_3_F_5" )
      I_Contact( "M_UD_3_F_6" )
      I_Contact( "M_UD_3_F_7" )
      I_Contact( "M_UD_3_B_1" )
      I_Contact( "M_UD_3_B_2" )
      I_Contact( "M_UD_3_B_3" )
      I_Contact( "M_UD_3_B_4" )
      I_Contact( "M_UD_3_B_5" )
      I_Contact( "M_UD_3_B_6" )
      I_Contact( "M_UD_3_B_7" )
      I_Contact( "UpDown".UD_3.I_SS_L )
   END_RUNG wire#w3
   RUNG wire#powerrail
      Contact( "M_UD_3_B_2" )
      wire#w4
      Coil( "UpDown".UD_3.O_Motor_B )
   END_RUNG
   RUNG wire#powerrail
      Contact( "M_UD_3_B_5" )
   END_RUNG wire#w4
   RUNG wire#powerrail
      Contact( "M_UD_3_B_7" )
   END_RUNG wire#w4
   // the same network as SCL:
   "UpDown".UD_3.O_Motor_F := "M_UD_3_F_3" OR "M_UD_3_F_7" OR "M_UD_3_F_5";
   "UpDown".UD_3.O_Motor_U := "M_UD_3_F_1" OR "M_UD_3_F_2" OR "M_UD_3_B_3" OR "M_UD_3_B_4";
   "UpDown".UD_3.O_Motor_D := "M_UD_3_F_4" OR "M_UD_3_B_1" OR (NOT "M_UD_3_F_1" AND NOT "M_UD_3_F_2" AND NOT "M_UD_3_F_3" AND NOT "M_UD_3_F_4" AND NOT "M_UD_3_F_5" AND NOT "M_UD_3_F_6" AND NOT "M_UD_3_F_7" AND NOT "M_UD_3_B_1" AND NOT "M_UD_3_B_2" AND NOT "M_UD_3_B_3" AND NOT "M_UD_3_B_4" AND NOT "M_UD_3_B_5" AND NOT "M_UD_3_B_6" AND NOT "M_UD_3_B_7" AND NOT "UpDown".UD_3.I_SS_L);
   "UpDown".UD_3.O_Motor_B := "M_UD_3_B_2" OR "M_UD_3_B_5" OR "M_UD_3_B_7";
END_REGION

REGION Network 242: Motor Control - updown 4
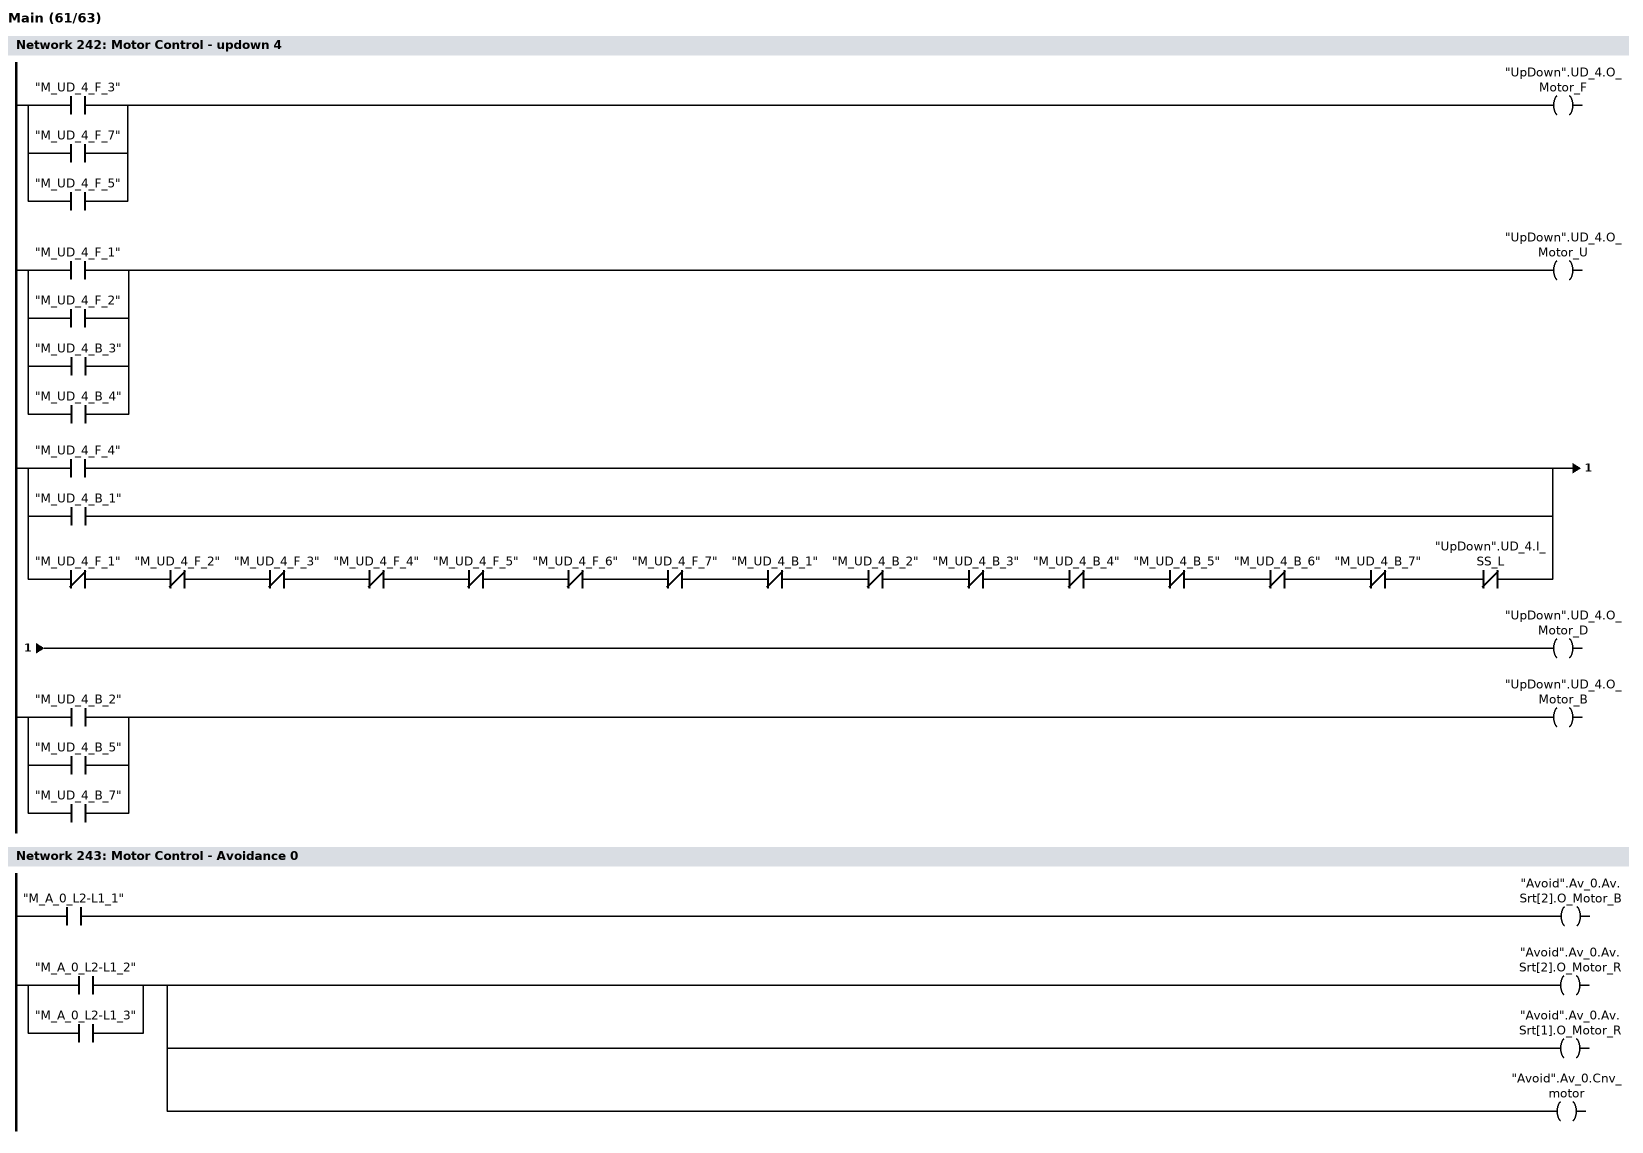
   RUNG wire#powerrail
      Contact( "M_UD_4_F_3" )
      wire#w1
      Coil( "UpDown".UD_4.O_Motor_F )
   END_RUNG
   RUNG wire#powerrail
      Contact( "M_UD_4_F_7" )
   END_RUNG wire#w1
   RUNG wire#powerrail
      Contact( "M_UD_4_F_5" )
   END_RUNG wire#w1
   RUNG wire#powerrail
      Contact( "M_UD_4_F_1" )
      wire#w2
      Coil( "UpDown".UD_4.O_Motor_U )
   END_RUNG
   RUNG wire#powerrail
      Contact( "M_UD_4_F_2" )
   END_RUNG wire#w2
   RUNG wire#powerrail
      Contact( "M_UD_4_B_3" )
   END_RUNG wire#w2
   RUNG wire#powerrail
      Contact( "M_UD_4_B_4" )
   END_RUNG wire#w2
   RUNG wire#powerrail
      Contact( "M_UD_4_F_4" )
      wire#w3
      Coil( "UpDown".UD_4.O_Motor_D )
   END_RUNG
   RUNG wire#powerrail
      Contact( "M_UD_4_B_1" )
   END_RUNG wire#w3
   RUNG wire#powerrail
      I_Contact( "M_UD_4_F_1" )
      I_Contact( "M_UD_4_F_2" )
      I_Contact( "M_UD_4_F_3" )
      I_Contact( "M_UD_4_F_4" )
      I_Contact( "M_UD_4_F_5" )
      I_Contact( "M_UD_4_F_6" )
      I_Contact( "M_UD_4_F_7" )
      I_Contact( "M_UD_4_B_1" )
      I_Contact( "M_UD_4_B_2" )
      I_Contact( "M_UD_4_B_3" )
      I_Contact( "M_UD_4_B_4" )
      I_Contact( "M_UD_4_B_5" )
      I_Contact( "M_UD_4_B_6" )
      I_Contact( "M_UD_4_B_7" )
      I_Contact( "UpDown".UD_4.I_SS_L )
   END_RUNG wire#w3
   RUNG wire#powerrail
      Contact( "M_UD_4_B_2" )
      wire#w4
      Coil( "UpDown".UD_4.O_Motor_B )
   END_RUNG
   RUNG wire#powerrail
      Contact( "M_UD_4_B_5" )
   END_RUNG wire#w4
   RUNG wire#powerrail
      Contact( "M_UD_4_B_7" )
   END_RUNG wire#w4
   // the same network as SCL:
   "UpDown".UD_4.O_Motor_F := "M_UD_4_F_3" OR "M_UD_4_F_7" OR "M_UD_4_F_5";
   "UpDown".UD_4.O_Motor_U := "M_UD_4_F_1" OR "M_UD_4_F_2" OR "M_UD_4_B_3" OR "M_UD_4_B_4";
   "UpDown".UD_4.O_Motor_D := "M_UD_4_F_4" OR "M_UD_4_B_1" OR (NOT "M_UD_4_F_1" AND NOT "M_UD_4_F_2" AND NOT "M_UD_4_F_3" AND NOT "M_UD_4_F_4" AND NOT "M_UD_4_F_5" AND NOT "M_UD_4_F_6" AND NOT "M_UD_4_F_7" AND NOT "M_UD_4_B_1" AND NOT "M_UD_4_B_2" AND NOT "M_UD_4_B_3" AND NOT "M_UD_4_B_4" AND NOT "M_UD_4_B_5" AND NOT "M_UD_4_B_6" AND NOT "M_UD_4_B_7" AND NOT "UpDown".UD_4.I_SS_L);
   "UpDown".UD_4.O_Motor_B := "M_UD_4_B_2" OR "M_UD_4_B_5" OR "M_UD_4_B_7";
END_REGION

REGION Network 243: Motor Control - Avoidance 0
   RUNG wire#powerrail
      Contact( "M_A_0_L2-L1_1" )
      Coil( "Avoid".Av_0.Av.Srt[2].O_Motor_B )
   END_RUNG
   RUNG wire#powerrail
      Contact( "M_A_0_L2-L1_2" )
      wire#w1
      Coil( "Avoid".Av_0.Av.Srt[2].O_Motor_R )
   END_RUNG
   RUNG wire#powerrail
      Contact( "M_A_0_L2-L1_3" )
   END_RUNG wire#w1
   RUNG wire#w1
      Coil( "Avoid".Av_0.Av.Srt[1].O_Motor_R )
   END_RUNG
   RUNG wire#w1
      Coil( "Avoid".Av_0.Cnv_motor )
   END_RUNG
   // the same network as SCL:
   "Avoid".Av_0.Av.Srt[2].O_Motor_B := "M_A_0_L2-L1_1";
   "Avoid".Av_0.Av.Srt[2].O_Motor_R := "M_A_0_L2-L1_2" OR "M_A_0_L2-L1_3";
   "Avoid".Av_0.Av.Srt[1].O_Motor_R := "M_A_0_L2-L1_2" OR "M_A_0_L2-L1_3";
   "Avoid".Av_0.Cnv_motor := "M_A_0_L2-L1_2" OR "M_A_0_L2-L1_3";
END_REGION

REGION Network 244: Motor Control - Avoidance 1to2
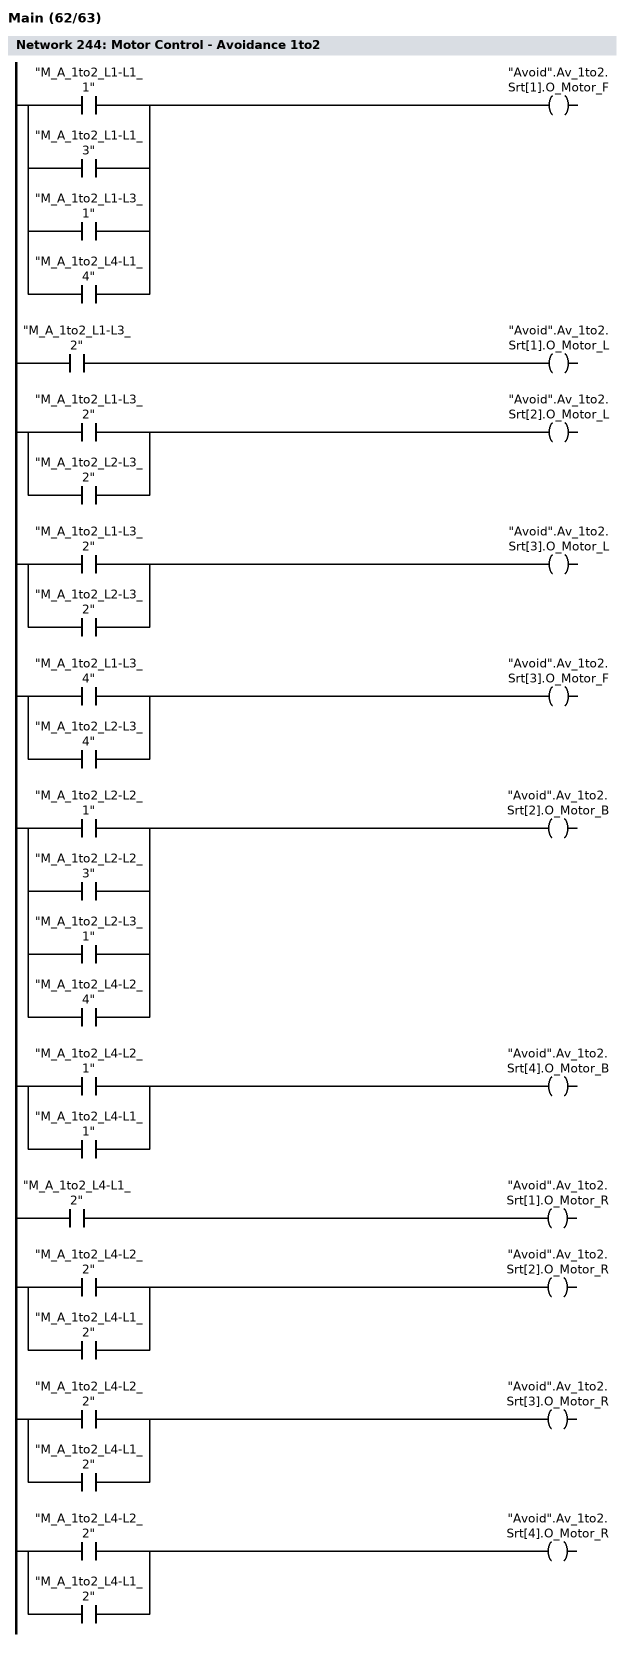
   RUNG wire#powerrail
      Contact( "M_A_1to2_L1-L1_1" )
      wire#w1
      Coil( "Avoid".Av_1to2.Srt[1].O_Motor_F )
   END_RUNG
   RUNG wire#powerrail
      Contact( "M_A_1to2_L1-L1_3" )
   END_RUNG wire#w1
   RUNG wire#powerrail
      Contact( "M_A_1to2_L1-L3_1" )
   END_RUNG wire#w1
   RUNG wire#powerrail
      Contact( "M_A_1to2_L4-L1_4" )
   END_RUNG wire#w1
   RUNG wire#powerrail
      Contact( "M_A_1to2_L1-L3_2" )
      Coil( "Avoid".Av_1to2.Srt[1].O_Motor_L )
   END_RUNG
   RUNG wire#powerrail
      Contact( "M_A_1to2_L1-L3_2" )
      wire#w2
      Coil( "Avoid".Av_1to2.Srt[2].O_Motor_L )
   END_RUNG
   RUNG wire#powerrail
      Contact( "M_A_1to2_L2-L3_2" )
   END_RUNG wire#w2
   RUNG wire#powerrail
      Contact( "M_A_1to2_L1-L3_2" )
      wire#w3
      Coil( "Avoid".Av_1to2.Srt[3].O_Motor_L )
   END_RUNG
   RUNG wire#powerrail
      Contact( "M_A_1to2_L2-L3_2" )
   END_RUNG wire#w3
   RUNG wire#powerrail
      Contact( "M_A_1to2_L1-L3_4" )
      wire#w4
      Coil( "Avoid".Av_1to2.Srt[3].O_Motor_F )
   END_RUNG
   RUNG wire#powerrail
      Contact( "M_A_1to2_L2-L3_4" )
   END_RUNG wire#w4
   RUNG wire#powerrail
      Contact( "M_A_1to2_L2-L2_1" )
      wire#w5
      Coil( "Avoid".Av_1to2.Srt[2].O_Motor_B )
   END_RUNG
   RUNG wire#powerrail
      Contact( "M_A_1to2_L2-L2_3" )
   END_RUNG wire#w5
   RUNG wire#powerrail
      Contact( "M_A_1to2_L2-L3_1" )
   END_RUNG wire#w5
   RUNG wire#powerrail
      Contact( "M_A_1to2_L4-L2_4" )
   END_RUNG wire#w5
   RUNG wire#powerrail
      Contact( "M_A_1to2_L4-L2_1" )
      wire#w6
      Coil( "Avoid".Av_1to2.Srt[4].O_Motor_B )
   END_RUNG
   RUNG wire#powerrail
      Contact( "M_A_1to2_L4-L1_1" )
   END_RUNG wire#w6
   RUNG wire#powerrail
      Contact( "M_A_1to2_L4-L1_2" )
      Coil( "Avoid".Av_1to2.Srt[1].O_Motor_R )
   END_RUNG
   RUNG wire#powerrail
      Contact( "M_A_1to2_L4-L2_2" )
      wire#w7
      Coil( "Avoid".Av_1to2.Srt[2].O_Motor_R )
   END_RUNG
   RUNG wire#powerrail
      Contact( "M_A_1to2_L4-L1_2" )
   END_RUNG wire#w7
   RUNG wire#powerrail
      Contact( "M_A_1to2_L4-L2_2" )
      wire#w8
      Coil( "Avoid".Av_1to2.Srt[3].O_Motor_R )
   END_RUNG
   RUNG wire#powerrail
      Contact( "M_A_1to2_L4-L1_2" )
   END_RUNG wire#w8
   RUNG wire#powerrail
      Contact( "M_A_1to2_L4-L2_2" )
      wire#w9
      Coil( "Avoid".Av_1to2.Srt[4].O_Motor_R )
   END_RUNG
   RUNG wire#powerrail
      Contact( "M_A_1to2_L4-L1_2" )
   END_RUNG wire#w9
   // the same network as SCL:
   "Avoid".Av_1to2.Srt[1].O_Motor_F := "M_A_1to2_L1-L1_1" OR "M_A_1to2_L1-L1_3" OR "M_A_1to2_L1-L3_1" OR "M_A_1to2_L4-L1_4";
   "Avoid".Av_1to2.Srt[1].O_Motor_L := "M_A_1to2_L1-L3_2";
   "Avoid".Av_1to2.Srt[2].O_Motor_L := "M_A_1to2_L1-L3_2" OR "M_A_1to2_L2-L3_2";
   "Avoid".Av_1to2.Srt[3].O_Motor_L := "M_A_1to2_L1-L3_2" OR "M_A_1to2_L2-L3_2";
   "Avoid".Av_1to2.Srt[3].O_Motor_F := "M_A_1to2_L1-L3_4" OR "M_A_1to2_L2-L3_4";
   "Avoid".Av_1to2.Srt[2].O_Motor_B := "M_A_1to2_L2-L2_1" OR "M_A_1to2_L2-L2_3" OR "M_A_1to2_L2-L3_1" OR "M_A_1to2_L4-L2_4";
   "Avoid".Av_1to2.Srt[4].O_Motor_B := "M_A_1to2_L4-L2_1" OR "M_A_1to2_L4-L1_1";
   "Avoid".Av_1to2.Srt[1].O_Motor_R := "M_A_1to2_L4-L1_2";
   "Avoid".Av_1to2.Srt[2].O_Motor_R := "M_A_1to2_L4-L2_2" OR "M_A_1to2_L4-L1_2";
   "Avoid".Av_1to2.Srt[3].O_Motor_R := "M_A_1to2_L4-L2_2" OR "M_A_1to2_L4-L1_2";
   "Avoid".Av_1to2.Srt[4].O_Motor_R := "M_A_1to2_L4-L2_2" OR "M_A_1to2_L4-L1_2";
END_REGION

REGION Network 245: Motor Control - Avoidance 2to3
